// TwinCAT 3 PLC project XtsTransport
// Title: XTS Transport
// Author: HAUD
// ProjectVersion: 4.01.02
// Description: . XTS_TRANSPORT_LAYER by Daniel Hauer
// ProgramVersion: 3.1.4026.26
// libraries:
//   Tc2_EtherCAT, * (Beckhoff Automation GmbH)
//   Tc2_Math, * (Beckhoff Automation GmbH)
//   Tc2_MC2, * (Beckhoff Automation GmbH)
//   Tc2_Standard, * (Beckhoff Automation GmbH)
//   Tc2_System, * (Beckhoff Automation GmbH)
//   Tc2_Utilities, * (Beckhoff Automation GmbH)
//   Tc2_XmlDataSrv, * (Beckhoff Automation GmbH)
//   Tc3_McCollisionAvoidance, * (Beckhoff Automation GmbH)
//   Tc3_McCoordinatedMotion, * (Beckhoff Automation GmbH)
//   Tc3_Module, * (Beckhoff Automation GmbH)
//   Tc3_XTS_Utility, * (Beckhoff Automation GmbH)
//   VisuDialogs, * (System)
// project tree:
//   APPLICATION/ GVL_APPLICATION.TcGVL (not stored), MAIN_APP.TcPOU, StationParameterExample.TcPOU, XTS_TRANSPORT_1.TcVIS (not stored)
//   APPLICATION/_config/ StationParameterExample.TcPOU (not stored)
//   APPLICATION/_types/Application/ E_APP_CHECK.TcDUT (not stored), E_APP_VARIANT.TcDUT (not stored), ST_APP_CTRL.TcDUT (not stored), ST_APP_STATE.TcDUT (not stored)
//   APPLICATION/_types/Collector/ E_PROCESS_CHECK.TcDUT (not stored), E_PROCESS_CTRL.TcDUT (not stored), E_PROCESS_STATE.TcDUT (not stored), fb_ProcessCollector.TcPOU (not stored), fb_StationCollector.TcPOU (not stored), I_ProcessCollector.TcIO (not stored), ST_PROCESS_CTRL.TcDUT (not stored), ST_PROCESS_STATE.TcDUT (not stored), T_PROCESS.TcDUT
//   APPLICATION/_types/ fb_ProcessConductor.TcPOU (not stored)
//   APPLICATION/_types/Instance/ E_INSTANCE.TcDUT (not stored), E_INSTANCE_CHECK.TcDUT (not stored), E_INSTANCE_CMD.TcDUT (not stored), E_INSTANCE_STATE.TcDUT (not stored), fb_Instance.TcPOU (not stored), ST_INSTANCE_CTRL.TcDUT (not stored), ST_INSTANCE_STATE.TcDUT (not stored)
//   APPLICATION/_types/LinkedList/ E_LIST_CHECK.TcDUT (not stored), E_LIST_CTRL.TcDUT (not stored), E_LIST_STATE.TcDUT (not stored), fb_Process_LinkedList.TcPOU (not stored), fb_Process_LinkedListCtrl.TcPOU (not stored), I_Process_LinkedList.TcIO (not stored), ST_LIST_CTRL.TcDUT (not stored), ST_LIST_NODE_DATA.TcDUT (not stored), ST_LIST_STATE.TcDUT (not stored), ST_PROCESS_DATA.TcDUT (not stored), ST_PROCESS_LIST_RESULT.TcDUT (not stored)
//   / GlobalTextList.TcGTLO, PlcTask.TcTTO
//   MAPPING/ MAPPING_XTS_in.TcPOU, MAPPING_XTS_out.TcPOU (not stored)
//   MAPPING/_types/ E_MAPPING_CHECK.TcDUT (not stored), U_APP_CTRL.TcDUT (not stored), U_APP_STATE.TcDUT (not stored), U_GEAR_DATA.TcDUT (not stored), U_INSTANCE_CTRL.TcDUT (not stored), U_INSTANCE_STATE.TcDUT (not stored), U_MOVER_CTRL.TcDUT (not stored), U_MOVER_INFO.TcDUT (not stored), U_MOVER_SELECTOR_CTRL.TcDUT (not stored), U_MOVER_SELECTOR_STATE.TcDUT (not stored), U_MOVER_STATE.TcDUT (not stored), U_MOVE_DATA.TcDUT (not stored), U_TICKET_LIST_CTRL.TcDUT (not stored), U_TICKET_LIST_DATA_INPUT.TcDUT (not stored), U_TICKET_LIST_DATA_OUTPUT.TcDUT (not stored), U_TICKET_LIST_STATE.TcDUT (not stored), U_XTS_STATION_CTRL.TcDUT (not stored), U_XTS_STATION_STATE.TcDUT (not stored), U_XTS_TRANSPORT_CTRL.TcDUT (not stored), U_XTS_TRANSPORT_STATE.TcDUT (not stored)
//   PLC_MOTION/_GVL/ PLC_CONSTANT.TcGVL
//   XTS_TRANSPORT/CaGroup/ FB_CaGroup.TcPOU (not stored), I_XtsTransport_CaGroup.TcIO (not stored)
//   XTS_TRANSPORT/CaGroup/types/ E_CA_GROUP_STATE.TcDUT, E_GROUP_CHECK.TcDUT, ST_GROUP_INFO.TcDUT
//   XTS_TRANSPORT/ GVL_XTS.TcGVL (not stored), GVL_XTS_CONSTANTS.TcGVL, GVL_XTS_VERSION.TcGVL (not stored), MAIN_XTS.TcPOU (not stored)
//   XTS_TRANSPORT/Mover/ fb_Mover.TcPOU (not stored), fb_MoverCtrl.TcPOU (not stored), fb_MoverSelector.TcPOU (not stored), I_XtsTransport_Mover.TcIO (not stored)
//   XTS_TRANSPORT/Mover/types/ E_MOVER_CHECK.TcDUT, E_MOVER_CTRL.TcDUT, E_MOVER_SELECTOR.TcDUT, E_MOVER_STATE.TcDUT, ST_GEAR_DATA.TcDUT, ST_MOVER_CTRL.TcDUT, ST_MOVER_INFO.TcDUT, ST_MOVER_SELECTOR_CTRL.TcDUT, ST_MOVER_SELECTOR_STATE.TcDUT, ST_MOVER_STATE.TcDUT, ST_MOVE_DATA.TcDUT
//   XTS_TRANSPORT/Xpu/ fb_Xpu.TcPOU (not stored), fb_XpuCtrl.TcPOU (not stored), I_XtsTransport_Xpu.TcIO (not stored)
//   XTS_TRANSPORT/Xpu/types/ E_XPU_CHECK.TcDUT, E_XPU_CTRL.TcDUT, E_XPU_INIT.TcDUT, E_XPU_STATE.TcDUT, ST_XPU_CTRL.TcDUT, ST_XPU_INFO.TcDUT, ST_XPU_STATE.TcDUT
//   XTS_TRANSPORT/XtsStation/ fb_StationGearInPos.TcPOU (not stored), fb_StationProcess.TcPOU (not stored), I_XtsTransport_Station.TcIO (not stored)
//   XTS_TRANSPORT/XtsStation/types/ E_STATION_CHECK.TcDUT, E_STATION_CTRL.TcDUT, E_STATION_GEAR_DISTANCE_AXIS.TcDUT, E_STATION_STATE.TcDUT, E_STATION_TYPE.TcDUT, fb_StationBase.TcPOU (not stored), fb_Station_LinkedList.TcPOU (not stored), I_Station_LinkedList.TcIO (not stored), ST_STATION_CTRL.TcDUT, ST_STATION_GEAR_PARAMETER.TcDUT, ST_STATION_LIST_RESULT.TcDUT, ST_STATION_MOVER_DATA.TcDUT, ST_STATION_PARAMETER.TcDUT, ST_STATION_STATE.TcDUT, T_NEST_OFFSET.TcDUT
//   XTS_TRANSPORT/XtsTransportUnit/ fb_TransportUnit.TcPOU (not stored)
//   XTS_TRANSPORT/XtsTransportUnit/types/ E_XTS_TRANSPORT_CHECK.TcDUT, E_XTS_TRANSPORT_CTRL.TcDUT, E_XTS_TRANSPORT_STATE.TcDUT, ST_XTS_TRANSPORT_CTRL.TcDUT, ST_XTS_TRANSPORT_STATE.TcDUT
//   XTS_TRANSPORT/_Visualization/ GROUP_VISU.TcVIS, MOVER_VISU.TcVIS, SELECTOR_VISU.TcVIS, STATION_VISU.TcVIS, Visualization Manager.TcVMO (not stored), XPU_VISU.TcVIS, XTS_TRANSPORT.TcVIS (not stored)
//   XTS_TRANSPORT/_Visualization/textlists/ TL_E_CTRL_MOVER.TcTLO, TL_E_CTRL_STATION.TcTLO, TL_E_CTRL_TRANSPORT.TcTLO, TL_E_CTRL_XPU.TcTLO, TL_E_MOVER_SELECTOR.TcTLO (not stored)
//   XTS_TRANSPORT/_Visualization/types/ ST_XPU_STRINGS.TcDUT, T_MOVER_SELECTOR.TcVIS
//   _MSG/class/ fb_LocalTime.TcPOU (not stored), fb_MessageData.TcPOU (not stored), fb_MessageDataCtrl.TcPOU
//   _MSG/ f_MessageSet.TcPOU (not stored), GVL_MSG_AXIS.TcGVL (not stored), GVL_MSG_XTS.TcGVL, I_MessageData.TcIO
//   _MSG/types/ e_Device.TcDUT, E_MessageType.TcDUT, E_MESSAGE_BATCH.TcDUT, E_MESSAGE_CHECK.TcDUT, E_MESSAGE_CTRL.TcDUT, E_MESSAGE_FLOW.TcDUT, E_MESSAGE_STATE.TcDUT, e_Subdevice.TcDUT, ST_Message.TcDUT, ST_MESSAGE_CTRL.TcDUT, ST_MESSAGE_STATE.TcDUT, TL_E_MESSAGETYPE.TcTLO
//   _types/ E_CHECK_STATE.TcDUT (not stored), E_PROGRESS.TcDUT (not stored), f_GetProgress.TcPOU (not stored), f_GetState.TcPOU (not stored), T_PROCESS.TcDUT (not stored)
//   _XML/Configuration/ fb_Configuration.TcPOU (not stored), I_Configuration_Station.TcIO (not stored)
//   _XML/Configuration/types/ ST_Configuration.TcDUT
//   _XML/ fb_XmlBase.TcPOU (not stored)
//   _XML/PositionOffsets/ fb_MoverPositionOffsetData.TcPOU (not stored)
//   _XML/PositionOffsets/types/ ST_MOVER_OFFSETS.TcDUT
//   _XML/types/ E_DATA_CHECK.TcDUT, E_DATA_CTRL.TcDUT, E_DATA_STATE.TcDUT, fb_XmlRead.TcPOU, fb_XmlWrite.TcPOU, ST_DATA_CTRL.TcDUT, ST_DATA_STATE.TcDUT
// (motion and I/O tree: see PLC project externcontrol)
// real-time tasks:
//   TASK XTS Task 1: cycle T#250us, priority 1, ADS port 350
//   TASK XTS Task 2: cycle T#250us, priority 3, ADS port 352
//   TASK PlcTask: cycle T#1ms, priority 15, ADS port 353
//   TASK Job Task: cycle default, priority 32
// variable links:
//   ExternControl/ExternControl Instance <-> XtsTransport/XtsTransport Instance
//     PlcTask Inputs/MAIN_APP.eInitXtsTransport <-> PlcTask Outputs/MAIN_APP.eInit
//     PlcTask Inputs/MAPPING_in.StationState.byState <-> PlcTask Outputs/MAPPING_XTS_out.StationState.byState
//     PlcTask Inputs/MAPPING_in.TransportState.byState <-> PlcTask Outputs/MAPPING_XTS_out.TransportState.byState
//     PlcTask Outputs/MAPPING_out.StationControl.byCtrl <-> PlcTask Inputs/MAPPING_XTS_in.StationControl.byCtrl
//     PlcTask Outputs/MAPPING_out.TransportControl.byCtrl <-> PlcTask Inputs/MAPPING_XTS_in.TransportControl.byCtrl
//   XtsTransport/XtsTransport Instance <-> NC-Task 1/Axes/Mover Axis 1
//     PlcTask Inputs/GVL_XTS.AxisRefMover[1].NcToPlc <-> Outputs/ToPlc
//     PlcTask Outputs/GVL_XTS.AxisRefMover[1].PlcToNc <-> Inputs/FromPlc
//   XtsTransport/XtsTransport Instance <-> NC-Task 1/Axes/Mover Axis 10
//     PlcTask Inputs/GVL_XTS.AxisRefMover[10].NcToPlc <-> Outputs/ToPlc
//     PlcTask Outputs/GVL_XTS.AxisRefMover[10].PlcToNc <-> Inputs/FromPlc
//   XtsTransport/XtsTransport Instance <-> NC-Task 1/Axes/Mover Axis 11
//     PlcTask Inputs/GVL_XTS.AxisRefMover[11].NcToPlc <-> Outputs/ToPlc
//     PlcTask Outputs/GVL_XTS.AxisRefMover[11].PlcToNc <-> Inputs/FromPlc
//   XtsTransport/XtsTransport Instance <-> NC-Task 1/Axes/Mover Axis 12
//     PlcTask Inputs/GVL_XTS.AxisRefMover[12].NcToPlc <-> Outputs/ToPlc
//     PlcTask Outputs/GVL_XTS.AxisRefMover[12].PlcToNc <-> Inputs/FromPlc
//   XtsTransport/XtsTransport Instance <-> NC-Task 1/Axes/Mover Axis 13
//     PlcTask Inputs/GVL_XTS.AxisRefMover[13].NcToPlc <-> Outputs/ToPlc
//     PlcTask Outputs/GVL_XTS.AxisRefMover[13].PlcToNc <-> Inputs/FromPlc
//   XtsTransport/XtsTransport Instance <-> NC-Task 1/Axes/Mover Axis 14
//     PlcTask Inputs/GVL_XTS.AxisRefMover[14].NcToPlc <-> Outputs/ToPlc
//     PlcTask Outputs/GVL_XTS.AxisRefMover[14].PlcToNc <-> Inputs/FromPlc
//   XtsTransport/XtsTransport Instance <-> NC-Task 1/Axes/Mover Axis 15
//     PlcTask Inputs/GVL_XTS.AxisRefMover[15].NcToPlc <-> Outputs/ToPlc
//     PlcTask Outputs/GVL_XTS.AxisRefMover[15].PlcToNc <-> Inputs/FromPlc
//   XtsTransport/XtsTransport Instance <-> NC-Task 1/Axes/Mover Axis 16
//     PlcTask Inputs/GVL_XTS.AxisRefMover[16].NcToPlc <-> Outputs/ToPlc
//     PlcTask Outputs/GVL_XTS.AxisRefMover[16].PlcToNc <-> Inputs/FromPlc
//   XtsTransport/XtsTransport Instance <-> NC-Task 1/Axes/Mover Axis 17
//     PlcTask Inputs/GVL_XTS.AxisRefMover[17].NcToPlc <-> Outputs/ToPlc
//     PlcTask Outputs/GVL_XTS.AxisRefMover[17].PlcToNc <-> Inputs/FromPlc
//   XtsTransport/XtsTransport Instance <-> NC-Task 1/Axes/Mover Axis 18
//     PlcTask Inputs/GVL_XTS.AxisRefMover[18].NcToPlc <-> Outputs/ToPlc
//     PlcTask Outputs/GVL_XTS.AxisRefMover[18].PlcToNc <-> Inputs/FromPlc
//   XtsTransport/XtsTransport Instance <-> NC-Task 1/Axes/Mover Axis 19
//     PlcTask Inputs/GVL_XTS.AxisRefMover[19].NcToPlc <-> Outputs/ToPlc
//     PlcTask Outputs/GVL_XTS.AxisRefMover[19].PlcToNc <-> Inputs/FromPlc
//   XtsTransport/XtsTransport Instance <-> NC-Task 1/Axes/Mover Axis 2
//     PlcTask Inputs/GVL_XTS.AxisRefMover[2].NcToPlc <-> Outputs/ToPlc
//     PlcTask Outputs/GVL_XTS.AxisRefMover[2].PlcToNc <-> Inputs/FromPlc
//   XtsTransport/XtsTransport Instance <-> NC-Task 1/Axes/Mover Axis 20
//     PlcTask Inputs/GVL_XTS.AxisRefMover[20].NcToPlc <-> Outputs/ToPlc
//     PlcTask Outputs/GVL_XTS.AxisRefMover[20].PlcToNc <-> Inputs/FromPlc
//   XtsTransport/XtsTransport Instance <-> NC-Task 1/Axes/Mover Axis 21
//     PlcTask Inputs/GVL_XTS.AxisRefMover[21].NcToPlc <-> Outputs/ToPlc
//     PlcTask Outputs/GVL_XTS.AxisRefMover[21].PlcToNc <-> Inputs/FromPlc
//   XtsTransport/XtsTransport Instance <-> NC-Task 1/Axes/Mover Axis 22
//     PlcTask Inputs/GVL_XTS.AxisRefMover[22].NcToPlc <-> Outputs/ToPlc
//     PlcTask Outputs/GVL_XTS.AxisRefMover[22].PlcToNc <-> Inputs/FromPlc
//   XtsTransport/XtsTransport Instance <-> NC-Task 1/Axes/Mover Axis 23
//     PlcTask Inputs/GVL_XTS.AxisRefMover[23].NcToPlc <-> Outputs/ToPlc
//     PlcTask Outputs/GVL_XTS.AxisRefMover[23].PlcToNc <-> Inputs/FromPlc
//   XtsTransport/XtsTransport Instance <-> NC-Task 1/Axes/Mover Axis 24
//     PlcTask Inputs/GVL_XTS.AxisRefMover[24].NcToPlc <-> Outputs/ToPlc
//     PlcTask Outputs/GVL_XTS.AxisRefMover[24].PlcToNc <-> Inputs/FromPlc
//   XtsTransport/XtsTransport Instance <-> NC-Task 1/Axes/Mover Axis 25
//     PlcTask Inputs/GVL_XTS.AxisRefMover[25].NcToPlc <-> Outputs/ToPlc
//     PlcTask Outputs/GVL_XTS.AxisRefMover[25].PlcToNc <-> Inputs/FromPlc
//   XtsTransport/XtsTransport Instance <-> NC-Task 1/Axes/Mover Axis 26
//     PlcTask Inputs/GVL_XTS.AxisRefMover[26].NcToPlc <-> Outputs/ToPlc
//     PlcTask Outputs/GVL_XTS.AxisRefMover[26].PlcToNc <-> Inputs/FromPlc
//   XtsTransport/XtsTransport Instance <-> NC-Task 1/Axes/Mover Axis 27
//     PlcTask Inputs/GVL_XTS.AxisRefMover[27].NcToPlc <-> Outputs/ToPlc
//     PlcTask Outputs/GVL_XTS.AxisRefMover[27].PlcToNc <-> Inputs/FromPlc
//   XtsTransport/XtsTransport Instance <-> NC-Task 1/Axes/Mover Axis 28
//     PlcTask Inputs/GVL_XTS.AxisRefMover[28].NcToPlc <-> Outputs/ToPlc
//     PlcTask Outputs/GVL_XTS.AxisRefMover[28].PlcToNc <-> Inputs/FromPlc
//   XtsTransport/XtsTransport Instance <-> NC-Task 1/Axes/Mover Axis 3
//     PlcTask Inputs/GVL_XTS.AxisRefMover[3].NcToPlc <-> Outputs/ToPlc
//     PlcTask Outputs/GVL_XTS.AxisRefMover[3].PlcToNc <-> Inputs/FromPlc
//   XtsTransport/XtsTransport Instance <-> NC-Task 1/Axes/Mover Axis 4
//     PlcTask Inputs/GVL_XTS.AxisRefMover[4].NcToPlc <-> Outputs/ToPlc
//     PlcTask Outputs/GVL_XTS.AxisRefMover[4].PlcToNc <-> Inputs/FromPlc
//   XtsTransport/XtsTransport Instance <-> NC-Task 1/Axes/Mover Axis 5
//     PlcTask Inputs/GVL_XTS.AxisRefMover[5].NcToPlc <-> Outputs/ToPlc
//     PlcTask Outputs/GVL_XTS.AxisRefMover[5].PlcToNc <-> Inputs/FromPlc
//   XtsTransport/XtsTransport Instance <-> NC-Task 1/Axes/Mover Axis 6
//     PlcTask Inputs/GVL_XTS.AxisRefMover[6].NcToPlc <-> Outputs/ToPlc
//     PlcTask Outputs/GVL_XTS.AxisRefMover[6].PlcToNc <-> Inputs/FromPlc
//   XtsTransport/XtsTransport Instance <-> NC-Task 1/Axes/Mover Axis 7
//     PlcTask Inputs/GVL_XTS.AxisRefMover[7].NcToPlc <-> Outputs/ToPlc
//     PlcTask Outputs/GVL_XTS.AxisRefMover[7].PlcToNc <-> Inputs/FromPlc
//   XtsTransport/XtsTransport Instance <-> NC-Task 1/Axes/Mover Axis 8
//     PlcTask Inputs/GVL_XTS.AxisRefMover[8].NcToPlc <-> Outputs/ToPlc
//     PlcTask Outputs/GVL_XTS.AxisRefMover[8].PlcToNc <-> Inputs/FromPlc
//   XtsTransport/XtsTransport Instance <-> NC-Task 1/Axes/Mover Axis 9
//     PlcTask Inputs/GVL_XTS.AxisRefMover[9].NcToPlc <-> Outputs/ToPlc
//     PlcTask Outputs/GVL_XTS.AxisRefMover[9].PlcToNc <-> Inputs/FromPlc
//   XtsTransport/XtsTransport Instance <-> NC-Task 1/Objects/Group1 (CA Group)
//     PlcTask Inputs/GVL_XTS.CaGroupRef.NcToPlc/CA <-> Group Outputs/ToPLC
//     PlcTask Outputs/GVL_XTS.CaGroupRef.PlcToNc/CA <-> Group Inputs/FromPLC

CONFIGURATION XtsTransport
    RESOURCE PLC ON TwinCAT3
        TASK PlcTask(INTERVAL := T#1ms, PRIORITY := 15);
        PROGRAM MAPPING_in WITH PlcTask : MAPPING_in;
        PROGRAM MAIN WITH PlcTask : MAIN;
        PROGRAM MAPPING_out WITH PlcTask : MAPPING_out;
    END_RESOURCE
END_CONFIGURATION

// ---- APPLICATION/_types/Collector/T_PROCESS.TcDUT
TYPE T_PROCESS : DWORD; END_TYPE

// ---- XTS_TRANSPORT/CaGroup/types/E_CA_GROUP_STATE.TcDUT
// {attribute 'qualified_only'}
// {attribute 'strict'}
{attribute 'to_string'}
TYPE E_CA_GROUP_STATE :
(
  // replicated from MC_GROUP_STATE for getting to_string() functionality
	mcGroupStateInvalid   :=0, 
  mcGroupStateDisabled  :=1, 
  mcGroupStateStandby   :=2, 
  mcGroupStateMoving    :=3, 
  mcGroupStateStopping  :=4, 
  mcGroupStateErrorStop :=5, 
  mcGroupStateHoming    :=6, 
  mcGroupStateNotReady  :=7, 
  mcGroupStateSuspended :=8 
)UINT;
END_TYPE

// ---- XTS_TRANSPORT/CaGroup/types/E_GROUP_CHECK.TcDUT
{attribute 'qualified_only'}
{attribute 'to_string'}
TYPE E_GROUP_CHECK :
(
  NULL,
  REFERENCE_GROUP_REF_INVALID := 9000,
  REFERENCE_AXIS_REF_INVALID,
  REFERENCE_CTRL_INVALID,
  REFERENCE_STATE_INVALID,
  REFERENCE_MOVER_ITF_INVALID,
  REFERENCE_XPU_INFO_INVALID,

  CHECK_DONE              := 10000
)UINT;
END_TYPE

// ---- XTS_TRANSPORT/CaGroup/types/ST_GROUP_INFO.TcDUT
TYPE ST_GROUP_INFO :
STRUCT
  GroupStatusValid,
  GroupStatusBusy,
  GroupMoving, 
  GroupHoming, 
  GroupErrorStop, 
  GroupNotReady, 
  GroupStandby, 
  GroupStopping,
 
  GroupDisabled, 
  AllAxesStanding, 
  ConstantVelocity, 
  Accelerating, 
  Decelerating, 
  InPosition, 
  GroupError					  : BIT; 

  GroupErrorId					: UDINT;

  AxisCount      				: UDINT;
  AxisCountEnabled      : UDINT;

  {attribute 'displaymode':='hex'}
  CaGroupOID            : OTCID;

  CaGroupState          : E_CA_GROUP_STATE;
END_STRUCT
END_TYPE

// ---- XTS_TRANSPORT/Mover/types/E_MOVER_CHECK.TcDUT
{attribute 'qualified_only'}
{attribute 'strict'}
{attribute 'to_string'}
TYPE E_MOVER_CHECK :
(
  NULL,
  MOVER_ID_INVALID := 9000,
  REFERENCE_AXIS_REF_INVALID,
  REFERENCE_LAST_POSITION_INVALID,
  REFERENCE_LAST_GAP_INVALID,
  REFERENCE_INFO_INVALID,

  REFERENCE_CTRL_INVALID  := 9100,
  REFERENCE_STATE_INVALID,
  REFERENCE_GEAR_DATA_INVALID,
  REFERENCE_MOVE_DATA_INVALID,
  REFERENCE_MOVER_ITF_INVALID,

  CHECK_DONE  := 10_000
)UINT;
END_TYPE

// ---- XTS_TRANSPORT/Mover/types/E_MOVER_CTRL.TcDUT
{attribute 'qualified_only'}
{attribute 'strict'}
{attribute 'to_string'}
TYPE E_MOVER_CTRL :
(
  MOVER_NULL,               // initial value at startup, used for change of order or retrigger
  MOVER_ENABLE,             // sets MC_Power.Enable
  MOVER_DISABLE,            // removes MC_Power.Enable
  MOVER_MOVE_TO_POS,        // modulo absolute positioning with MC_MoveAbsolute, InTargetPosition check
  MOVER_MOVE_TO_POS_CA,     // modulo absolute positioning with MC_MoveAbsoluteCA, InTargetPosition check
  MOVER_SEND_TO_POS_CA,     // modulo absolute positioning with MC_MoveAbsoluteCA, done after moving ReleaseDistance
  MOVER_HALT,               // halts mover; by use of MC_Halt mover is set passive in CA group
  MOVER_GEAR_IN,            // GearIn for mover in standstill

  MOVER_GEAR_IN_POS_CA,     // GearInPosCA of mover; when FB_GearInPosCa is InSync --> order is done; check SyncDistance yourself and release mover with e_mover_order.mover_SendToPos
  MOVER_GEAR_OUT,           // gear out for mover
  MOVER_RESET,              // MC_RESET for mover
  MOVER_INFO                // used to display MoverInfo in ST_MOVER_SELECTOR_STATE.Info
)UINT;
END_TYPE

// ---- XTS_TRANSPORT/Mover/types/E_MOVER_SELECTOR.TcDUT
{attribute 'qualified_only'}
{attribute 'strict'}
{attribute 'to_string'}
TYPE E_MOVER_SELECTOR :
(
	SELECT_MOVER_INDEX,
  SELECT_MOVER_AXIS_ID
);
END_TYPE

// ---- XTS_TRANSPORT/Mover/types/E_MOVER_STATE.TcDUT
{attribute 'qualified_only'}
{attribute 'to_string'}
TYPE E_MOVER_STATE :
(
  MOVER_NULL,               // initial value at startup, used for change of order or retrigger
  MOVER_ENABLE,             // sets MC_Power.Enable
  MOVER_DISABLE,            // removes MC_Power.Enable
  MOVER_MOVE_TO_POS,        // modulo absolute positioning with MC_MoveAbsolute, InTargetPosition check
  MOVER_MOVE_TO_POS_CA,     // modulo absolute positioning with MC_MoveAbsoluteCA, InTargetPosition check
  MOVER_SEND_TO_POS_CA,     // modulo absolute positioning with MC_MoveAbsoluteCA, done after moving ReleaseDistance
  MOVER_HALT,               // halts mover; by use of MC_Halt mover is set passive in CA group
  MOVER_GEAR_IN,            // GearIn for mover in standstill

  MOVER_GEAR_IN_POS_CA,     // GearInPosCA of mover; when FB_GearInPosCa is InSync --> order is done; check SyncDistance yourself and release mover with e_mover_order.mover_SendToPos
  MOVER_GEAR_OUT,           // gear out for mover
  MOVER_RESET,              // MC_RESET for mover
  MOVER_INFO
)UINT;
END_TYPE

// ---- XTS_TRANSPORT/Mover/types/ST_GEAR_DATA.TcDUT
{attribute 'pack_mode' := '2'}
TYPE ST_GEAR_DATA :
STRUCT
  rDeltaToMasterPos       : LREAL;
  rModuloSyncPosSlave     : LREAL;
  rMasterStartDistance    : LREAL;
  rGearNumerator          : LREAL;
  iGearDenumerator        : USINT  := 1;
END_STRUCT
END_TYPE

// ---- XTS_TRANSPORT/Mover/types/ST_MOVER_CTRL.TcDUT
{attribute 'pack_mode' := '2'}
TYPE ST_MOVER_CTRL :
STRUCT
  Cmd             : E_MOVER_CTRL;  // order to execute on mover
END_STRUCT
END_TYPE

// ---- XTS_TRANSPORT/Mover/types/ST_MOVER_INFO.TcDUT
{attribute 'pack_mode' := '2'}
TYPE ST_MOVER_INFO :
STRUCT
  bMoverEnabled           : BIT;    // Axis[i].Status.ControlLoopClosed
  bMoverError             : BIT;    // Axis[i].Status.Error
  bMoverCoupled           : BIT;    // Axis[i].Status.Coupled OR _fbGearInPosCa[i].InSync
  bMoverStandstill        : BIT;    // Axis[i].Status.NotMoving
  bMoverAvoidingCollision : BIT;    // Axis[i].NcToPlc.StateDWord2.0
  bMoverInTarget          : BIT;    // Axis[i].NcToPlc.ActPos == rLastSetPos[i]

  rModuloActPos           : LREAL;  // Axis[i].NcToPlc.ModuloActPos
  rAbsActPos              : LREAL;  // Axis[i].NcToPlc.ActPos
  rAbsTargetPos           : LREAL;  // rLastSetPos[i]
  rModuloTargetPos        : LREAL;  // Tc2_Math.LMOD(_rLastSetPos[i], _RailLength)

  nErrorId                : UDINT;
END_STRUCT
END_TYPE

// ---- XTS_TRANSPORT/Mover/types/ST_MOVER_SELECTOR_CTRL.TcDUT
TYPE ST_MOVER_SELECTOR_CTRL :
STRUCT
  Selector      : E_MOVER_SELECTOR; // select by array Index OR AXIS_REF.NcToPlc.AxisId 
  Mover         : UINT;             // array Index OR AXIS_REF.NcToPlc.AxisId
  Control       : ST_MOVER_CTRL;    // mover control struct, put motion command in here

  Data          : ST_MOVE_DATA;     // write your movement parameters
  //Gear          : ST_GEAR_DATA;     // write your gearing parameters
END_STRUCT
END_TYPE

// ---- XTS_TRANSPORT/Mover/types/ST_MOVER_SELECTOR_STATE.TcDUT
TYPE ST_MOVER_SELECTOR_STATE :
STRUCT
  MoverIndex  : UINT;
  AxisId      : UDINT;
  State       : ST_MOVER_STATE;

  Info        : ST_MOVER_INFO;
END_STRUCT
END_TYPE

// ---- XTS_TRANSPORT/Mover/types/ST_MOVER_STATE.TcDUT
{attribute 'pack_mode' := '2'}
TYPE ST_MOVER_STATE :
STRUCT
  State           : E_MOVER_STATE;  // ST_MOVER_CTRL.Cmd with added E_PROGRESS
  MasterId        : USINT;            // mirror NC AxisId of Master axis
END_STRUCT
END_TYPE

// ---- XTS_TRANSPORT/Mover/types/ST_MOVE_DATA.TcDUT
{attribute 'pack_mode' := '2'}
TYPE ST_MOVE_DATA :
STRUCT
  // HAUD 2024 03 14
  // some init data added for example
  rPos            : LREAL :=   2275.0;
  rVelo           : LREAL :=    500.0;
  rAcc            : LREAL :=   5000.0;
  rJerk           : LREAL := 500000.0;
  rGap            : LREAL :=    100.0;
  rOverride       : LREAL :=    100.0;
  rDelta          : LREAL :=      0.05;
  rDistance       : LREAL :=     25.0;
END_STRUCT
END_TYPE

// ---- XTS_TRANSPORT/Xpu/types/E_XPU_CHECK.TcDUT
{attribute 'qualified_only'}
{attribute 'to_string'}
TYPE E_XPU_CHECK :
(
  INIT_CHECK,
  INIT_CHECK_ERROR,
  START_CHECK,
  XPU_INSTANCE_NULL,
  XPU_RAIL_LENGTH,
  GROUP_RAIL_LENGTH,
  RAIL_LENGTH_COMPARE,
  GROUP_NOT_CONFIGURED,
  GROUP_OID_MISMATCH,

  MOVER_COUNT             := 10,
  MOVER_COUNT_ZERO,
  MOVER_COUNT_NOT_EQUAL,

  PROCESSING_UNIT_POSITIONS_VALID         := 20,
  PROCESSING_UNIT_GET_DATA_EXCEED,

  MOVER_ID_STANDARD       := 30,
  MOVER_ID_SIMULATION,
  MOVER_ID_DETECTION_MODE,
  MOVER_ID_DETECTION_VALID,
  MOVER_ID_DETECTION_DC_LINK,
  MOVER_ID_DETECTION_BUSY,
  MOVER_ID_DETECTION_IDLE,
  MOVER_ID_DETECTION_STATE,
  MOVER_ID_MULTIPLE_NOT_SUPPORTED,

  POINTER_CHECK           := 90,
  POINTER_NULL_CTRL,
  POINTER_NULL_STATE,

  CHECK_DONE      := 10_000
)UINT;
END_TYPE

// ---- XTS_TRANSPORT/Xpu/types/E_XPU_CTRL.TcDUT
{attribute 'strict'}
TYPE E_XPU_CTRL :
(
  XTS_CMD_NULL,
  XTS_CMD_INIT                  := 10,
  //XTS_CMD_READ_STN_CONFIG       := 20,
  XTS_IDLE                      := 30
)UINT;
END_TYPE

// ---- XTS_TRANSPORT/Xpu/types/E_XPU_INIT.TcDUT
{attribute 'to_string'}
TYPE E_XPU_INIT :
(
	INIT_START,
  INIT_ENVIRONMENT_OID            := 10,
  INIT_INFO_SERVER_ITF,
  INIT_INFO_SERVER_STATION_COUNT,
  INIT_INFO_SERVER_STATION_OID,
  INIT_CA_GROUP_OID               := 20,
  INIT_CA_GROUP_GET_OID,
  INIT_CA_GROUP_CHECK_OID,
  INIT_CA_GROUP_COM,
  INIT_PARAMETERSET_COUNT,
  INIT_PARAMETERSET_OID,
  INIT_PARAMETERSET_COM,
  INIT_PARAMETERSET_COM_INIT,
  INIT_PARAMETERSET_COM_NEXT,
  INIT_PROCESSING_UNIT_COM        := 30,
  INIT_PROCESSING_UNIT_COM_INIT,
  INIT_PROCESSING_UNIT_PART_COUNT,
  INIT_PROCESSING_UNIT_PART_OID,
  INIT_PROCESSING_UNIT_TRACK_COUNT,
  INIT_PROCESSING_UNIT_TRACK_OID,
  INIT_PROCESSING_UNIT_MOVER_COUNT,
  INIT_PROCESSING_UNIT_MOVER_OID,
  INIT_PROCESSING_UNIT_TASK_COUNT,
  INIT_PROCESSING_UNIT_TASK_OID,
  INIT_TRACK_COM                  := 50,
  INIT_TRACK_COM_INIT,
  INIT_PART_COM                   := 60,
  INIT_PART_COM_INIT,
  INIT_PART_MODULE_COUNT,
  INIT_PART_MODULE_OID,
  INIT_PART_MODULE_COM,
  INIT_PART_MODULE_COM_INIT,
  INIT_PART_MODULE_COM_NEXT,
  INIT_MOVER_COM                  := 70,
  INIT_MOVER_COM_INIT,
  INIT_MOVER_COM_NEXT,
  INIT_NCT_CONTROLLER_OID         := 80,
  INIT_NCT_CONTROLLER_COM,
  INIT_NCT_CONTROLLER_COM_INIT,
  INIT_NCT_BASE_UNIT_COUNT,
  INIT_NCT_BASE_UNIT_ITF,
  INIT_NCT_BASE_UNIT_NEXT,
  INIT_DATA_GET                   := 90,
  INIT_DATA_CHECK,
  INIT_DONE                       := 100
)UINT;
END_TYPE

// ---- XTS_TRANSPORT/Xpu/types/E_XPU_STATE.TcDUT
{attribute 'to_string'}
TYPE E_XPU_STATE :
(
  XTS_NULL,
  XTS_INVALID,
  XTS_INIT                      := 10,    // initialize XPU
  XTS_STATION_INFO_READ         := 20,    // get Station information from Xpu
  XTS_IDLE                      := 30
)UINT;
END_TYPE

// ---- XTS_TRANSPORT/Xpu/types/ST_XPU_CTRL.TcDUT
{attribute 'pack_mode' := '2'}
TYPE ST_XPU_CTRL :
STRUCT
  Cmd             : E_XPU_CTRL;
END_STRUCT
END_TYPE

// ---- XTS_TRANSPORT/Xpu/types/ST_XPU_INFO.TcDUT
{attribute 'pack_mode' := '2'}
TYPE ST_XPU_INFO :
STRUCT
  AllPositionsValid   : BIT;
  IdDetectionError    : BIT;
  IdDetectionValid    : BIT;
  IdDetectionActive   : BIT;

  OperationMode       : UINT;

  IdDetectionMode           : UINT;
  MoverPositionAssignement  : UINT;

  nDetectedAxisCount  : UINT;
  nExpectedAxisCount  : UINT;

  nParameterSetCount  : UINT;
  nModuleCount        : UINT;
  rRailLength         : LREAL;
END_STRUCT
END_TYPE

// ---- XTS_TRANSPORT/Xpu/types/ST_XPU_STATE.TcDUT
{attribute 'pack_mode' := '2'}
TYPE ST_XPU_STATE :
STRUCT
  Init            : E_XPU_INIT;
  State           : E_XPU_STATE;
  Check           : E_XPU_CHECK;  // cyclic check result
  DcLink          : BIT;          // power all motor modules is ON
END_STRUCT
END_TYPE

// ---- XTS_TRANSPORT/XtsStation/types/E_STATION_CHECK.TcDUT
{attribute 'qualified_only'}
{attribute 'strict'}
{attribute 'to_string'}
TYPE E_STATION_CHECK :
(
	CHECK_NULL,
  STATION_ID_INVALID := 9000,
  REFERENCE_CTRL_INVALID,
  REFERENCE_STATE_INVALID,
  REFERENCE_LIST_ITF_INVALID,
  REFERENCE_MOVER_ITF_INVALID,
  REFERENCE_MOVER_OFFSET_INVALID,
  REFERENCE_PARAMETER_INVALID,
  REFERENCE_MOVER_AXIS_REF_INVALID,

  REFERENCE_MASTER_AXIS_REF_INVALID,
  REFERENCE_GEAR_DATA_INVALID,
  REFERENCE_GEAR_PARAMETER_INVALID,

  CHECK_DONE    := 10_000
);
END_TYPE

// ---- XTS_TRANSPORT/XtsStation/types/E_STATION_CTRL.TcDUT
{attribute 'qualified_only'}
{attribute 'strict'}
{attribute 'to_string'}
TYPE E_STATION_CTRL :
(
  STATION_CTRL_NULL,              // nothing happens here
	STATION_INIT            := 1,   // hard reset of station, list is cleared
  STATION_DISABLE         := 10,  // 
  STATION_ENABLE,                 // 

  STATION_MOVER_ENTER     := 20,  // mover may enter station
  STATION_MOVER_ENTER_RETRY,      // retry after E_STATION_STATE.STATION_ERROR_INFEED_ERROR
  STATION_MOVER_SEND,             // do not enter, send to E_STATION_STATE.STATION_MOVER_OUT

  STATION_PROCESS_START   := 30,  // double handshake with extern
  STATION_PROCESS_DONE,           // single handshake with extern
  STATION_PROCESS_NEST_SKIP,

  STATION_MOVER_OUT       := 50,  // mover may leave station now; ticket for mover is checked here (ST_STATION_CTRL.nTargetStation)
  STATION_MOVER_OUT_RETRY,        // retry after E_STATION_STATE.STATION_ERROR_OUTFEED_ERROR

  STATION_MOVER_GONE      := 60   // mover has left station, last handshake station is empty

)USINT;
END_TYPE

// ---- XTS_TRANSPORT/XtsStation/types/E_STATION_GEAR_DISTANCE_AXIS.TcDUT
{attribute 'qualified_only'}
{attribute 'strict'}
{attribute 'to_string'}
TYPE E_STATION_GEAR_DISTANCE_AXIS :
(
  // which axis nSync distance is checked for termination of GearInPosCA.
  // after nSync distance the station does a regular outfeed to target station
	FOLLOW_THE_MASTER,
  FOLLOW_THE_SLAVE
)UINT;
END_TYPE

// ---- XTS_TRANSPORT/XtsStation/types/E_STATION_STATE.TcDUT
{attribute 'qualified_only'}
{attribute 'to_string'}
TYPE E_STATION_STATE :
(
	STATION_NO_INIT,                // startup state after power on, first cycle Init of station, switches to INIT when done

  STATION_INIT,                   // CONTINUE to DISABLE
                                  // State.MoverId deleted

  STATION_DISABLE         := 10,  // + CTRL.STATION_ENABLE  --> CONTINUE to DETECT_MOVER 
                                  // station is empty, no mover is handled, check enable from ctrl

  STATION_ENABLE,                 // init of work vars, check enable from ctrl

  STATION_DETECT_MOVER,           // (QueueCount > 0)       --> CONTINUE to MOVER_ENTER

  STATION_MOVER_ENTER     := 20,  // + CTRL.MOVER_ENTER     --> CONTINUE to PROCESS_START
                                  // + CTRL.MOVER_SEND      --> CONTINUE to MOVER_OUT
                                  // mover asking for entry

  STATION_MOVER_IN_TARGET,        // (MoveToPos==TRUE)      --> CONTINUE to PROCESS_START
                                  // mover is moving to PosWait + PosStop[_nNest]

  STATION_PROCESS_START   := 30,  // + CTRL.PROCESS_START   --> CONTINUE to PROCESS_START
                                  // + CTRL.PROCESS_DONE    --> CONTINUE to CHECK
                                  // wait until process started

  STATION_PROCESS_DONE,           // + CTRL.PROCESS_DONE    --> CONTINUE to CHECK
                                  // wait until process done

  STATION_CHECK           := 40,  // check for next nest in mask, 
                                  // (mask<>0) --> CHECK_NEST
                                  // (mask==0) --> MOVER_OUT

  STATION_CHECK_NEST,             // + CTRL.MOVER_ENTER     --> CONTINUE to MOVER_IN_TARGET
                                  // get next nest position

  STATION_MOVER_OUT       := 50,  // + CTRL.MOVER_OUT       --> CONTINUE to MOVER_RELEASE
                                  // mover asking to leave

  STATION_MOVER_RELEASE,          // (MoverSendToPos==TRUE) --> CONTINUE to MOVER_GONE
                                  // mover is released + check if release distance is passed

  STATION_MOVER_WRITE_TARGET,     // worker state to write mover ticket

  STATION_MOVER_GONE      := 60,  // + CTRL.MOVER_GONE      --> CONTINUE to INIT
                                  // mover out of station, enter mover in target station list


  STATION_ERROR_NULL      := 127,
  STATION_ERROR_LIST_GET_HEAD_FAULT,    // fatal error in linked list, must never occurr, must be debugged
  STATION_ERROR_LIST_REMOVE_HEAD_FAULT, // fatal error in linked list, must never occurr, must be debugged
  STATION_ERROR_LIST_ADD_TAIL_FAULT,    // fatal error in linked list, must never occurr, must be debugged

  STATION_ERROR_LIST_STATION_ID_WRONG,  // ticket data in Queue contains wrong Station Id, can be overruled by ctrl

  STATION_ERROR_LIST_MOVER_ID_INVALID,  // fatal error in ticket data, MoverId is out of range, must be fixed by ctrl, must be debugged

  STATION_ERROR_INFEED_ERROR,           // motion error during movement, retry must be triggered by ctrl
  STATION_ERROR_OUTFEED_ERROR,          // motion error during movement, retry by ctrl OR leave by ctrl

  STATION_ERROR_OUTFEED_TARGET_INVALID, // ticket data for nTargetStation is not plausible, can be fixed by ctrl

  STATION_ERROR_FATAL     := 255 // the thing that must not be, all fatal errors end up here
)USINT;
END_TYPE

// ---- XTS_TRANSPORT/XtsStation/types/E_STATION_TYPE.TcDUT
{attribute 'qualified_only'}
{attribute 'strict'}
{attribute 'to_string'}
TYPE E_STATION_TYPE :
(
	INVALID,
  STATION_PROCESS,      // default station with/without process
  STATION_GEAR_IN_POS   // GearInPos station for flying saw with MasterAxis
)USINT;
END_TYPE

// ---- XTS_TRANSPORT/XtsStation/types/ST_STATION_CTRL.TcDUT
{attribute 'pack_mode' := '2'}
TYPE ST_STATION_CTRL :
STRUCT
  Cmd             : E_STATION_CTRL;
  {attribute 'displaymode':='bin'}
  nMask           : BYTE;           // nest mask for sending mover to next station
  nTargetStation  : USINT;          // where to next?
  rOffset         : REAL;           // optional offset for mover in target station when leaving sending station; 
                                    // use case: position correction of workpiece on wpc by vision
END_STRUCT
END_TYPE

// ---- XTS_TRANSPORT/XtsStation/types/ST_STATION_GEAR_PARAMETER.TcDUT
TYPE ST_STATION_GEAR_PARAMETER :
STRUCT
  eDistance           : E_STATION_GEAR_DISTANCE_AXIS; // follow which leader?
  rSyncDistance       : LREAL := 100.0;               // synchrone distance while the mover is geared in
  rMinDistanceToSync  : LREAL := 100.0;               // minimum distance for mover to get nSync with the Master
END_STRUCT
END_TYPE

// ---- XTS_TRANSPORT/XtsStation/types/ST_STATION_LIST_RESULT.TcDUT
TYPE ST_STATION_LIST_RESULT :
STRUCT
  wState    : WORD;   // wState == 0 --> all ok
  nIndex    : ULINT;
  stData    : ST_STATION_MOVER_DATA;  // copy of list entry
END_STRUCT
END_TYPE

// ---- XTS_TRANSPORT/XtsStation/types/ST_STATION_MOVER_DATA.TcDUT
{attribute 'pack_mode' := '2'}
TYPE ST_STATION_MOVER_DATA :
STRUCT
  nMoverId        : USINT;  // who am I?  !! MUST be correct !! - movement to base position sets everything in order, DO NOT manipulate!
  nTargetStation  : USINT;  // where shall I be? used for double checking with StationId at infeed of mover into station

  {attribute 'displaymode':='bin'}
  nMask           : BYTE;   // how many of you are there? (1 = default, no action required)

  rOffset         : REAL;   // offset for use in work flow !! added to static mover offset for every nest(bit) in nMask!!
END_STRUCT
END_TYPE

// ---- XTS_TRANSPORT/XtsStation/types/ST_STATION_PARAMETER.TcDUT
TYPE ST_STATION_PARAMETER :
STRUCT
  eType             : E_STATION_TYPE := 1;  // StationProcess or StationGearInPos
  sText             : STRING(80);           // only description
  rPosWait          : REAL;                 // start of station, 
                                            // a sending station is using this value 
                                            // to send mover to

  rReleaseDistance  : REAL;                 // distance mover has to travel (from ActPos) 
                                            // in order for station to go back to disable

  rGap              : REAL;
  rVelo             : REAL;
  rAccDec           : REAL;
  rJerk             : REAL;

  // how many nests (stop positions) mover has to stop at (1 = default)
  nConfiguredStopCount  : USINT := 1; // 1-8 --> NestMask = BYTE

  // mover stop position in station, relative to rPosWait!!
  rPosStop          : ARRAY[1..8] OF LREAL;
END_STRUCT
END_TYPE

// ---- XTS_TRANSPORT/XtsStation/types/ST_STATION_STATE.TcDUT
{attribute 'pack_mode' := '2'}
TYPE ST_STATION_STATE :
STRUCT
  State           : E_STATION_STATE;
  {attribute 'displaymode':='bin'}
  nMask           : BYTE;
  nMoverId        : USINT;
  rMoverModPos    : LREAL;            // modulo position of detected mover
  nQueue          : USINT;            // queue count for station
END_STRUCT
END_TYPE

// ---- XTS_TRANSPORT/XtsStation/types/T_NEST_OFFSET.TcDUT
TYPE T_NEST_OFFSET : ARRAY[1..MAX_MOVER]        OF
                     ARRAY[1..MAX_STATION_NEST] OF LREAL;
END_TYPE

// ---- XTS_TRANSPORT/XtsTransportUnit/types/E_XTS_TRANSPORT_CHECK.TcDUT
{attribute 'qualified_only'}
{attribute 'to_string'}
TYPE E_XTS_TRANSPORT_CHECK :
(
  // info for cyclic checks
  INIT_CHECK,
  START_CHECK,    // check cycle start
  XPU_INIT,       // Xpu: initialization


  // errors in fb_TransportUnit.Check()
  POINTER_CHECK           := 9000,
  POINTER_NULL_CTRL,

  POINTER_NULL_STATE,
  POINTER_NULL_XPU_CTRL,

  POINTER_NULL_XPU_STATE,
  POINTER_NULL_XPU_INFO,

  POINTER_NULL_GROUP_ITF,
  POINTER_NULL_GROUP_INFO,

  POINTER_NULL_MOVER,
  POINTER_NULL_MOVER_ITF,

  POINTER_NULL_MOVER_INFO,
  POINTER_NULL_MOVER_LAST_POS,
  POINTER_NULL_MOVER_LAST_GAP,

  POINTER_NULL_STATION_START,
  POINTER_NULL_STATION_ITF,
  POINTER_NULL_STATION_CONTROL,
  POINTER_NULL_STATION_STATE,
  POINTER_NULL_STATION_CTRL_ITF,

  DONE_CHECK              := 10000
)UINT;
END_TYPE

// ---- XTS_TRANSPORT/XtsTransportUnit/types/E_XTS_TRANSPORT_CTRL.TcDUT
{attribute 'strict'}
{attribute 'to_string'}
TYPE E_XTS_TRANSPORT_CTRL :
(
  CMD_NULL,
  CMD_INIT                  := 10,  // Xpu, Group, Mover initialization: clear errors, clear group, check Xpu data, check mover detection
  CMD_IDLE,

  CMD_MOVER_ENABLE          := 20,  // all mover are enabled, checked for ControlLoopClosed
  CMD_MOVER_DISABLE,                // all mover are disabled, no axis in CaGroup: no error, any axis in CaGroup: group error
  CMD_MOVER_HALT_CA,                // all movers are stopped with MC_HaltCA[]. ONLY use if all movers are in CA group
  CMD_MOVER_STOP,

  CMD_GROUP_CLEAR           := 30,  // halt all movers, clear errors, remove all movers from group, clear group
  CMD_GROUP_BUILD,                  // add all movers to group
  CMD_GROUP_ENABLE,                 // group with movers is enabled
  CMD_GROUP_STOP,                   // moving CA Group is stopped

  CMD_TRANSPORT_START       := 40,  // move all mover[i] to start position
  CMD_TRANSPORT_RESTART             // move all mover[i] to LastPosition[i]

)UINT;
END_TYPE

// ---- XTS_TRANSPORT/XtsTransportUnit/types/E_XTS_TRANSPORT_STATE.TcDUT
{attribute 'to_string'}
TYPE E_XTS_TRANSPORT_STATE :
(
  TRANSPORT_NULL,
  TRANSPORT_INVALID,
  TRANSPORT_INIT            := 10,  // Xpu, Group, Mover initialization: init TcCOM objects, clear errors, clear group, check Xpu data, check mover detection
  TRANSPORT_IDLE,                   // cyclic check for errors, check Xpu data

  TRANSPORT_MOVER_ENABLE    := 20,  // all mover are enabled, checked for ControlLoopClosed
  TRANSPORT_MOVER_DISABLE,          // all mover are disabled
  TRANSPORT_MOVER_HALT_CA,          // all mover standstill
  TRANSPORT_MOVER_STOP,

  TRANSPORT_GROUP_CLEAR     := 30,  // halt all movers, clear errors, remove all movers from group, clear group
  TRANSPORT_GROUP_BUILD,            // add all movers to group
  TRANSPORT_GROUP_ENABLE,           // group with movers is enabled
  TRANSPORT_GROUP_STOP,             // CaGroup Stop, CaGroup Reset, All movers halt

  TRANSPORT_START           := 40,  // move all mover[i] to start position
  TRANSPORT_RESTART                 // move all mover[i] to LastPosition[i]
)UINT;
END_TYPE

// ---- XTS_TRANSPORT/XtsTransportUnit/types/ST_XTS_TRANSPORT_CTRL.TcDUT
{attribute 'pack_mode' := '2'}
TYPE ST_XTS_TRANSPORT_CTRL :
STRUCT
  Cmd       : E_XTS_TRANSPORT_CTRL;
END_STRUCT
END_TYPE

// ---- XTS_TRANSPORT/XtsTransportUnit/types/ST_XTS_TRANSPORT_STATE.TcDUT
{attribute 'pack_mode' := '2'}
TYPE ST_XTS_TRANSPORT_STATE :
STRUCT
  State         : E_XTS_TRANSPORT_STATE;  // combined value of state and result(e_progress); (hint: extract state value by mod division)
  Check         : E_XTS_TRANSPORT_CHECK;

  XpuState      : ST_XPU_STATE;
  XpuInfo       : ST_XPU_INFO;
  GroupInfo     : ST_GROUP_INFO; 
END_STRUCT
END_TYPE

// ---- XTS_TRANSPORT/_Visualization/types/ST_XPU_STRINGS.TcDUT
TYPE ST_XPU_STRINGS :
STRUCT
  sXpuState       ,
  sXpuResult      ,
  sXpuCyclicCheck ,
  sXpuOpMode      ,
  sXpuMoverId_DetectionMode,
  sXpuMoverPosAssignement : STRING(30) := 'NULL';
END_STRUCT
END_TYPE

// ---- _MSG/types/e_Device.TcDUT
{attribute 'to_string'}
TYPE e_Device :
(
  Device_Null,                  // NULL               - not to be used
  Device_Main,                  // MAIN(PRG)          - reserved for MAIN(PRG)
  Device_MainAxis,              // MAIN_AXIS(PRG)     - reserved for MAIN_AXIS(PRG)
  Device_Nci,                   // NCI(PRG)           - reserved for NCI(PRG)
  Device_Cam,                   // CAM(PRG            - reserved for CAM(PRG)
  Device_Functions,             // FUNCTIONS(PRG)     - reserved for FUNCTIONS(PRG)
  Device_FlyingSaw,             // FLYING_SAW(PRG)    - reserved for FLYING_SAW(PRG)
  Device_MainApplication,       // MAIN_APP(PRG)      - reserved for MAIN_APP(PRG)

  Device_MoverSelector,         // single mover interface for xts applications
  Device_ParameterSelector,     // fb_ParameterSelector can only exist once in a project.
  Device_Configuration,         // fb_Configuration can handle multiple files therefore only one instance is required
  Device_XmlData,               // generic XML Data (e.g. persistent data)
  Device_Utilities,             // service calls to anyone you may want to talk to, the main intent is to get XPU and TcXtsIo data to the application side

  General           :=  1000,
  CaGroup           :=  2000,
  Xpu               :=  3000,
  XpuCtrl           :=  4000,
  Mover             :=  5000,
  MoverCtrl         :=  6000,
  XtsTransportUnit  :=  7000,
  XfcTriggerBox     :=  8000,
  XfcTouchProbe     :=  9000,
  XtsStation        := 10000,

  Camming           := 11000,
  NciChannel        := 12000,
  NciChannelCtrl    := 13000,
  Axis              := 14000,
  XfcAxis           := 15000,

  // txt file logging LOG_FILE_METRICS
  MetricsXts        := 16000,   //entries from xts Metrics are written into dedicated txt file (see f_MessageSet, here's the diverter)
  MetricsAxis       := 17000,   //entries from PLC_MOTION Metrics are written into dedicated txt file

  // txt file logging LOG_FILE_APP
  Process           := 20000,   // entries from process are written into dedicated txt file.
  ProcessListCtrl   := 21000,
  TicketListCtrl    := 22000,

  Application       := 30000,   // entries from application are written into dedicated txt file.


  // txt file logging LOG_FILE_PRODUCT - this is for you to use
  DataProduct       := 40000
)UDINT;
END_TYPE

// ---- _MSG/types/E_MessageType.TcDUT
{attribute 'strict'}
{attribute 'to_string'}
TYPE E_MessageType :
(
  //-----------------------------------------------------
  //-----------------------------------------------------
  //  message system:
  //  - errors are always calling f_MessageSet()
  //  - errors are always entered into its list
  //
  //  - message severity is set by this enum (like everywhere else)
  //
  //  - message frequency is set by this enum
  //    - IF you get above 50 stations, 
  //      writing to the file system takes time:
  //
  //    Batch: switching on metrics (> Empty) must not add cpu load, 
  //      --> so do not clutter here
  //
  //    Info:  regular flow of information (>Error / >Warning) 
  //           must not add significant cpu load, 
  //      --> so do not clutter here
  //
  //    Verbose and above:
  //    --> for small systems (< 96 mover, < 50 stations) 
  //        you may switch it on for everybody, 
  //        files get big quickly ;-)
  //
  //    --> switch on during test phase for a handful of stations
  //
  //    --> high detail logging always and for everybody
  //    --> we need somebody who transfers data more quickly
  //      --> I can offer a .NET(C#) ADS tool which collects the list.
  //          .NET application then pushes to database
  //-----------------------------------------------------
  //-----------------------------------------------------
  eMessageEmpty,    // he who is without bounds may speak
  eMessageBatch,    // he who counts words, counts numbers (Batch started, Next in Batch, Batch done)
  eMessageError,    // mine, your(')s, anybody's, let the numbers tell you
  eMessageWarning,  // I told you so
  eMessageInfo,     // A long time ago in a galaxy far, far away...
  eMessageVerbose,  // He talks a lot, doesn't he?; Yeah! He's very knowledgeable.
  eMessageSentient  // Keep them out of bright light, Don't get them wet, do not feed them after midnight!! No matter how much they beg!!
)DINT;
END_TYPE

// ---- _MSG/types/E_MESSAGE_BATCH.TcDUT
{attribute 'qualified_only'}
{attribute 'strict'}
{attribute 'to_string'}
TYPE E_MESSAGE_BATCH :
(
	MSG_BATCH_NULL,
  MSG_BATCH_JOB_STARTED,
  MSG_BATCH_NEXT_IN_JOB,
  MSG_BATCH_JOB_DONE
)UINT;
END_TYPE

// ---- _MSG/types/E_MESSAGE_CHECK.TcDUT
{attribute 'qualified_only'}
{attribute 'strict'}
{attribute 'to_string'}
TYPE E_MESSAGE_CHECK :
(
  NULL,
  // 9000 --> here comes your error
  POINTER_INVALID             := 9000,
  POINTER_TIME_INVALID,
  POINTER_LIST_INVALID,
  POINTER_MSG_IDX_INVALID,
  POINTER_ERR_IDX_INVALID,
  POINTER_ROOT_FILE_INVALID,
  POINTER_ROOT_DIR_INVALID,
  POINTER_CTRL_INVALID,
  POINTER_STATE_INVALID,

  // 10000 --> here comes your man
  CHECK_DONE                        := 10000
)UINT;
END_TYPE

// ---- _MSG/types/E_MESSAGE_CTRL.TcDUT
{attribute 'qualified_only'}
{attribute 'strict'}
{attribute 'to_string'}
TYPE E_MESSAGE_CTRL :
(
	MSG_CTRL_NULL,
	MSG_CTRL_INIT   := 10,
  MSG_CTRL_IDLE   := 30,
  MSG_CTRL_WRITE  := 50
)UINT;
END_TYPE

// ---- _MSG/types/E_MESSAGE_FLOW.TcDUT
{attribute 'qualified_only'}
{attribute 'strict'}
{attribute 'to_string'}
TYPE E_MESSAGE_FLOW :
(
  MSG_FLOW_INIT,
  MSG_FLOW_ROOT                 := 10,
  MSG_FLOW_ROOT_CREATE,
  MSG_FLOW_ROOT_CREATE_BUSY,
  MSG_FLOW_FOLDER,
  MSG_FLOW_FOLDER_CREATE,
  MSG_FLOW_FOLDER_CREATE_BUSY,
  MSG_FLOW_FILE_CREATE_DONE,
  MSG_FLOW_LINE_START           := 100,
  MSG_FLOW_LINE_BUILD,
  MSG_FLOW_LINE_CHECK,
  MSG_FLOW_WRITE_FILE_BUSY      := 200,
  MSG_FLOW_WRITE_FILE_END,
  MSG_FLOW_WRITE_FILE_DONE      := 1000
)UINT;
END_TYPE

// ---- _MSG/types/E_MESSAGE_STATE.TcDUT
{attribute 'qualified_only'}
//{attribute 'strict'}
{attribute 'to_string'}
TYPE E_MESSAGE_STATE :
(
	MSG_STATE_NULL,
  MSG_STATE_INIT    := 10,
  MSG_STATE_IDLE    := 30,
  MSG_STATE_WRITE   := 50
)UINT;
END_TYPE

// ---- _MSG/types/e_Subdevice.TcDUT
{attribute 'strict'}
{attribute 'to_string'}
TYPE e_Subdevice :
(
  // sub device for message system
  General                 :=  0,
  MainInit,
  // Motion Control FB Instances
  fbPower,
  fbReset,
  fbResetSercos,
  fbHalt,
  fbStop,                 // 5
  fbHome,
  fbJog,
  fbMoveVelocity1,
  fbMoveVelocity2,
  fbMoveAbsolute1,        // 10
  fbMoveAbsolute2,
  fbMoveEndless,
  fbMovePtP,
  fbMoveVelo,
  fbSendToPos,

  // CA CollisionAvoidance FB instances
  // CA group fb instances
  fbCaGroup             := 30,
  fbMoveToPosCa,
  fbSendToAbsPosCa,
  fbSendToModuloPosCa,
  fbGearInPosCa,
  fbGroupAddAxis,
  fbGroupRemoveAxis,
  fbGroupDisable,
  fbGroupEnable,
  fbGroupErrorRead,
  fbGroupStatusRead,
  fbGroupReset,
  fbGroupStop,
  fbHaltCa,

  fbGearIn                := 50,
  fbGearOut,
  fbGearInMultiMaster,

  fbCamOutV2              := 80,
  fbCamInV2,
  fbCamScalingV2,
  fbCamInfoV2,
  fbReadMotionFunction,
  fbReadMotionFunctionPoint,
  fbReadMotionFunctionValues,
  fbWriteMotionFunction,
  fbWriteMotionFunctionPoint,
  fbSetOnlineChangeMode,

  fbReadParameter         := 100,
  fbReadBoolParameter,
  fbWriteParameter,
  fbWriteBoolParameter,
  fbWriteParameterPersistent,
  fbXmlRead,
  fbXmlWrite,
  fbCreateFolder,

  fbBuildGroup            := 200,
  fbClearGroup,
  fbLoadProg,
  fbResetItp,
  fbStartStopItp,
  fbEStopItp,             // 205
  fbStepOnAfterEStopItp,
  fbConfirmHskItp,
  fbDelDtgItp,
  fbNciFeedTablePreparation,
  fbNciFeedTable,         // 210
  fbReadLine,
  fbItpReadRParams,
  fbItpWriteRParams,
  Get_ItpState,
  Get_Error,              // 215


  XfcPositionAtTime       := 300,
  XfcTimeOfPosition,
  XfcTimeToPosition,
  XfcTimeToModuloPosition,
  XfcRecordedPosition,
  XfcTouchProbe,          // 305
  XfcTouchProbeEL1258,
  XfcTouchProbeOptions,
  XfcTriggerRef,
  XfcTriggerRef_MT,
  XfcEl1258Interface_MT,  // 310
  XfcRecordedPosition_MT,
  XfcTriggerOut,
  XfcTriggerStart,
  XfcSwitchOn_2252,
  XfcSwitchOff_2252,      // 315
  XfcInit,
  XfcLatchPosition,
  XfcWaitForPosition,

  AxisMode              := 1000,
  AxisControl,
  AxisStartUp,
  AxisCycle,
  AxisIdle,

  NciControl            := 2000,
  NciStartUp,
  NciCycle,
  NciIdle,

  FlyingSawControl      := 2100,
  FlyingSawStartUp,

  StationLinkedList     := 3000,
  StationInitList,
  StationAddHead,
  StationAddTail,
  StationGetHead,
  StationRemoveHeadValue,
  StationGearInDistanceToSync,
  StationGearInSyncStart,
  StationGearInSyncMove,
  StationGearInSyncEnd,
  StationCalcInfeedPosition,

  StationControl        := 4000,
  StationState, 

  Xpu_fbEnvironment     := 5000,
  Xpu_fbProcessingUnit,
  Xpu_fbXpuPart,
  Xpu_fbXpuTrack,
  Xpu_fbMc2CaGroup,
  Xpu_fbParameterSet,
  Xpu_fbNctController,

  Xpu_fbPartModules     := 5500,

  Xpu_fbMoverXpu        := 6000,

  Xpu_fbNctBaseUnit     := 6500,

  TransportUnit_General := 7000,
  TransportUnit_Restart := 7010,
  TransportUnit_Start,
  TransportUnit_XpuInit,
  TransportUnit_StationClearOutfeed,
  TransportUnit_GroupEnable,
  TransportUnit_GroupClear,
  TransportUnit_GroupBuild,
  TransportUnit_GroupStop,
  TransportUnit_MoverEnableAll,
  TransportUnit_MoverDisableAll,


  CamControl            := 8000,
  CamStartUp,
  CamCycle,

  Process_StationCollector    := 11000,
  Process_ProcessCollector    := 11100,
  Process_ProcessCollector_Init,
  Process_ProcessCollector_Cycle,
  Process_ProcessCollector_Control,

  Process_LinkedList_GetHead,
  Process_LinkedList_RemoveHead,
  Process_LinkedList_AddTail,
  Process_LinkedList_CheckData,
  Process_StationQueue_Check,

  Process_LinkedList_Com              := 11200,
  Process_LinkedList_Com_Init,
  Process_LinkedList_Com_Cmd,
  Process_LinkedList_Com_AddHead,
  Process_LinkedList_Com_AddTail,
  Process_LinkedList_Com_DelHead,
  Process_LinkedList_Com_DelTail,
  Process_LinkedList_Com_GetHead,
  Process_LinkedList_Com_GetTail,


  Instance_Command              := 12000,
  Instance_ProcessConductor,
  Instance_BufferInfeed,
  Instance_Infeed,
  Instance_BufferOutfeed,
  Instance_Outfeed,
  Instance_Sender_Buffer,

  Ticket_LinkedList_Ctrl        := 12100,
  Ticket_LinkedList_Com_Init,
  Ticket_LinkedList_Com_Cmd,
  Ticket_LinkedList_Com_AddHead,
  Ticket_LinkedList_Com_AddTail,
  Ticket_LinkedList_Com_DelHead,
  Ticket_LinkedList_Com_DelTail,
  Ticket_LinkedList_Com_GetHead,
  Ticket_LinkedList_Com_GetTail,
  

  Application                 := 13000,
  Application_Check,
  Application_Clear,
  Application_Cmd,
  Application_Disable,
  Application_Enable,
  Application_Finish,
  Application_Init,
  Application_Proceed,
  Application_Work,

  Utilities                   := 13100,
  Utilities_GetStationOnModule,
  Utilities_SetGlobalConstraints

)DINT;
END_TYPE

// ---- _MSG/types/ST_Message.TcDUT
TYPE ST_Message :
STRUCT
  eType         : e_MessageType;
  eDevice       : e_Device;
  eSubdevice    : e_SubDevice;
  {attribute 'displaymode':='hex'}
  iErrorNumber  : LINT;
  tTime         : STRING(24);
  sText         : STRING(127);
END_STRUCT
END_TYPE

// ---- _MSG/types/ST_MESSAGE_CTRL.TcDUT
TYPE ST_MESSAGE_CTRL :
STRUCT
  Cmd         : E_MESSAGE_CTRL;
END_STRUCT
END_TYPE

// ---- _MSG/types/ST_MESSAGE_STATE.TcDUT
TYPE ST_MESSAGE_STATE :
STRUCT
  State         : E_MESSAGE_STATE;  // as always... combined value of Cmd equivalent and e_progress
END_STRUCT
END_TYPE

// ---- _XML/Configuration/types/ST_Configuration.TcDUT
TYPE ST_Configuration :
STRUCT
  XtsStationParameter  : ARRAY[1..MAX_STATION] OF ST_STATION_PARAMETER;
END_STRUCT
END_TYPE

// ---- _XML/PositionOffsets/types/ST_MOVER_OFFSETS.TcDUT
TYPE ST_MOVER_OFFSETS :
STRUCT
  // static position offsets in stations
  PositionOffset      : ARRAY[1..MAX_STATION] OF T_NEST_OFFSET; // added to PosStop[] in XtsStation
END_STRUCT
END_TYPE

// ---- _XML/types/E_DATA_CHECK.TcDUT
{attribute 'qualified_only'}
{attribute 'strict'}
{attribute 'to_string'}
TYPE E_DATA_CHECK :
(
  NULL,
  REFERENCE_CTRL_INVALID  := 9000,
  REFERENCE_STATE_INVALID,

  POINTER_STATION_PARAMETER_INVALID := 9100,
  POINTER_MOVER_DISTANCES_INVALID,
  POINTER_MOVER_OFFSETS_INVALID,

  DONE_CHECK              := 10000
);
END_TYPE

// ---- _XML/types/E_DATA_CTRL.TcDUT
{attribute 'qualified_only'}
{attribute 'to_string'}
{attribute 'strict'}
TYPE E_DATA_CTRL :
(
  NULL,
	INIT  := 10,
  READ  := 20,
  WRITE := 30
)UINT;
END_TYPE

// ---- _XML/types/E_DATA_STATE.TcDUT
{attribute 'qualified_only'}
{attribute 'to_string'}
TYPE E_DATA_STATE :
(
	NULL,
  NO_EXIST,
  INIT        := 10,
  READ        := 20,
  WRITE       := 30
)UINT;
END_TYPE

// ---- _XML/types/ST_DATA_CTRL.TcDUT
{attribute 'pack_mode' := '2'}
TYPE ST_DATA_CTRL :
STRUCT
  Cmd       : E_DATA_CTRL;
END_STRUCT
END_TYPE

// ---- _XML/types/ST_DATA_STATE.TcDUT
{attribute 'pack_mode' := '2'}
TYPE ST_DATA_STATE :
STRUCT
  State       : E_DATA_STATE;
  Init        : E_PROGRESS;
END_STRUCT
END_TYPE

// ---- PLC_MOTION/_GVL/PLC_CONSTANT.TcGVL
//{attribute 'qualified_only'}
VAR_GLOBAL CONSTANT


  //-----------------------------------------------------------------------------
  // AXIS related limits
  //-----------------------------------------------------------------------------
  MAX_AXIS              : UINT    := 3;
  MAX_RETRY             : UINT    := 5;


  //-----------------------------------------------------------------------------
  // NCI related limits and *.nc standard folder
  //-----------------------------------------------------------------------------
{IF NOT defined (BSD)}
  NCI_DIR               : STRING  := 'C:\TwinCAT\Mc\Nci\';
{ELSE}
  NCI_DIR               : STRING  := '/usr/local/etc/TwinCAT/Mc/Nci/';
{END_IF}

{IF defined (NCI)}
  {info 'PLC_MOTION_LAYER: NCI'}
  NCI_ACTIVE            : BOOL    := TRUE;
  CONFIG_NAME           : STRING  := 'NCI_Spec_Ch_';
{ELSE}
  NCI_ACTIVE            : BOOL    := FALSE;
  CONFIG_NAME           : STRING  := 'NCI_NOT_ACTIVE';
{END_IF}

  MAX_NCI_CH            : UINT    := 1;

  MAX_PATH_STEPS        : UINT    := 5;
  MAX_MC_AXIS           : UINT    := 3;
  MAX_AUX_AXIS          : UINT    := 2;
  MAX_R_PARA            : UINT    := 10;


  //-----------------------------------------------------------------------------
  // CAMMING related limits
  //-----------------------------------------------------------------------------
{IF defined (CAM)}
  {info 'PLC_MOTION_LAYER: CAM'}
  CAM_ACTIVE                  : BOOL    := TRUE;
{ELSE}
  CAM_ACTIVE                  : BOOL    := FALSE;
{END_IF}

  MAX_CAM_CH                  : UINT    := 1;

  MAX_MOTION_FUNCTION_POINTS  : UINT    := 10;

  // HAUD
  // 17.07.2024
  // Start Implementation of Position Trigger function
  //  - Timestamp/position output
  //  - Latch DC time from input
  
  MAX_TRIGGER_BOX             : UINT := 12;
  MAX_TOUCH_PROBE             : UINT := 12;
  MAX_TRIGGER_COUNT           : UINT :=  4;
  MAX_MTI_CH                  : UINT :=  1; // MAX mti channel per EL terminal

{IF defined (XFC)}
  {info 'PLC_MOTION_LAYER: XFC'}
  XFC_ACTIVE                  : BOOL := TRUE;
{ELSE}
  XFC_ACTIVE                  : BOOL := FALSE;
{END_IF}

  // HAUD
  // 2026 05 28
  // Gear In Pos implementation for flying saw application 

{IF defined (SAW)}
  {info 'PLC_MOTION_LAYER: FLYING_SAW'}
  FLY_SAW_ACTIVE              : BOOL  := TRUE;
{ELSE}
  FLY_SAW_ACTIVE              : BOOL  := FALSE;
{END_IF}
END_VAR

// ---- XTS_TRANSPORT/GVL_XTS_CONSTANTS.TcGVL
//{attribute 'qualified_only'}
VAR_GLOBAL CONSTANT
//-----------------------------------------------------------------------------------------------------------------------------------------
//-----------------------------------------------------------------------------------------------------------------------------------------
//
//  HAUD 2026.03.15
//  - parameter list deleted (never used the parameter feature anyway), 
//    back to static global constants
//
//-----------------------------------------------------------------------------------------------------------------------------------------
//-----------------------------------------------------------------------------------------------------------------------------------------
//  Connections to XTS Utility Lib data: 
//  - suits this simple approach, 
//  - leaves you options to expand, 
//  - expansion and multiplication is not implemented here on purpose, 
//  - this project is designed to get the main ideas across, 
//  - setting up a matrix for multiple fb_Xpu instances with it, 
//    --> a second step you might want to organize from here; 
//        --> I leave the details up to you
//-----------------------------------------------------------------------------------------------------------------------------------------
//-----------------------------------------------------------------------------------------------------------------------------------------
  MAX_MOVER           : UINT    := TO_UINT(Tc3_XTS_Utility.TcIoXtsEnvironmentParameterList.MaxXtsMoversPerXpu);
  MAX_MODULE          : UINT    := TO_UINT(Tc3_XTS_Utility.TcIoXtsEnvironmentParameterList.MaxModulesPerPart);
  MAX_PART            : UINT    := TO_UINT(Tc3_XTS_Utility.TcIoXtsEnvironmentParameterList.MaxXtsPartsPerXpu);
  MAX_TRACK           : UINT    := TO_UINT(Tc3_XTS_Utility.TcIoXtsEnvironmentParameterList.MaxXtsTracksPerXpu);
  MAX_GROUP           : UINT    := TO_UINT(Tc3_XTS_Utility.TcIoXtsEnvironmentParameterList.MaxXtsCaGroup);

  MAX_INFO_SERVER     : UINT    := TO_UINT(Tc3_XTS_Utility.TcIoXtsEnvironmentParameterList.MaxXtsInfoServer);
  MAX_INFO_STATION    : UINT    := TO_UINT(Tc3_XTS_Utility.TcIoXtsEnvironmentParameterList.MaxXtsInfoStation);
  MAX_INFO_STOP_POS   : UINT    := TO_UINT(Tc3_XTS_Utility.TcIoXtsEnvironmentParameterList.MaxXtsStopPositionsPerStation);

  MAX_PARAMETER_SET   : UINT    := TO_UINT(Tc3_XTS_Utility.TcIoXtsEnvironmentParameterList.MaxXtsParameterSet);

  MAX_NCT_BASE_UNIT   : UINT    := TO_UINT(Tc3_XTS_Utility.TcIoXtsEnvironmentParameterList.MaxXtsNctBaseUnitInterfaces);
//-----------------------------------------------------------------------------------------------------------------------------------------
//-----------------------------------------------------------------------------------------------------------------------------------------
//  XTS_TRANSPORT_LAYER
//  - project constants you will have to adjust in order to build your transport logic
//-----------------------------------------------------------------------------------------------------------------------------------------
//-----------------------------------------------------------------------------------------------------------------------------------------
  MAX_STATION         : UINT    := 21;

  MAX_STATION_NEST    : UINT    := TO_UINT(SIZEOF(ST_STATION_STATE.nMask)*8);
  MAX_LIST_NODES      : UINT    := MAX_MOVER;
  MAX_MASTER          : UINT    := 1;
//-----------------------------------------------------------------------------------------------------------------------------------------
//-----------------------------------------------------------------------------------------------------------------------------------------
END_VAR

// ---- _MSG/GVL_MSG_XTS.TcGVL
{attribute 'qualified_only'}
VAR_GLOBAL CONSTANT
  //-----------------------------------------------------------------------------
  // file paths for message system
  //  - compiler define option WIN switches to Windows file paths
  //-----------------------------------------------------------------------------
{IF defined (WIN)}
  {info 'WIN folders'}
  LOG_DIR               : STRING  := 'C:\TwinCAT\#MsgFiles\';       // delimiter at the end is mandatory!!
  CON_DIR               : STRING  := 'C:\TwinCAT\#Configuration\';  // delimiter at the end is mandatory!!
{ELSE}
  {info 'BSD folders'}
  LOG_DIR               : STRING  := '/usr/local/etc/TwinCAT/#MsgFiles/';       // delimiter at the end is mandatory!!
  CON_DIR               : STRING  := '/usr/local/etc/TwinCAT/#Configuration/';  // delimiter at the end is mandatory!!
{END_IF}

  LOG_FILE              : STRING  := 'MSG_XtsTransport_';
  LOG_FILE_APP          : STRING  := 'MSG_Application_';
  LOG_FILE_METRIC       : STRING  := 'MSG_XtsTransportMetrics_';

  MAX_MESSAGE           : UINT    := 2000; // max entry in message list
END_VAR
VAR_GLOBAL
  //-----------------------------------------------------------------------------
  // Message System
  //  - Everybody uses f_MessageSet(ST_Message)
  //    - DECISION WHICH LIST IS MADE IN f_MessageSet !!
  //    - which list to use is determined by e_Device in your message
  //
  //  - MessageData instances are self sufficient and need only 
  //    datafield assignment for correct data-flow
  //
  //
  //-----------------------------------------------------------------------------
  //-----------------------------------------------------------------------------
  //-----------------------------------------------------------------------------
  // (ST_Message.eDevice := e_Device.Application)
  //----------------------------------------------------------------------------- 
  ApplicationMessageData          : fb_MessageDataCtrl;
  ApplicationMessageCtrl          : st_message_ctrl;
  ApplicationMessageState         : st_message_state;

  ApplicationMessages             : ARRAY[1..MAX_MESSAGE] OF ST_Message;
  MessageApplicationIndex         : UINT := 0; // message index for higher layers (grouping, Instances, etc.)
  MessageApplicationError         : UINT := 0; // error counter for higher learning
  //-----------------------------------------------------------------------------
  //-----------------------------------------------------------------------------
  // (ST_Message.eDevice := from Device_Null to XfcAxis)
  //-----------------------------------------------------------------------------
  TransportMessageData            : fb_MessageDataCtrl;
  TransportMessageCtrl            : st_message_ctrl;
  TransportMessageState           : st_message_state;

  TransportMessages               : ARRAY[1..MAX_MESSAGE] OF ST_Message;
  MessageTransportIndex           : UINT := 0; // message index for base layer
  MessageTransportError           : UINT := 0; // error counter for base layer
  //-----------------------------------------------------------------------------
  //-----------------------------------------------------------------------------
  // (ST_Message.eDevice := e_Device.Metrics)
  //-----------------------------------------------------------------------------
  MetricsMessageData              : fb_MessageDataCtrl;
  MetricsMessageCtrl              : st_message_ctrl;
  MetricsMessageState             : st_message_state;

  MetricsMessages                 : ARRAY[1..MAX_MESSAGE] OF ST_Message;
  MessageMetricsIndex             : UINT := 0; // message index for metrics data
  MessageMetricsError             : UINT := 0; // error counter for metrics data
  //-----------------------------------------------------------------------------
  //-----------------------------------------------------------------------------
  // (ST_Message.eDevice := e_Device.ProductData)
  //-----------------------------------------------------------------------------
  ProductMessageData              : fb_MessageDataCtrl;   // This is for you
  ProductMessageCtrl              : st_message_ctrl;
  ProductMessageState             : st_message_state;

  ProductMessages                 : ARRAY[1..MAX_MESSAGE] OF ST_Message;
  MessageProductIndex             : UINT := 0; // message index for your product data
  MessageProductError             : UINT := 0; // error counter for your product data
  //-----------------------------------------------------------------------------
  //-----------------------------------------------------------------------------
  fbLocalTime                     : fb_LocalTime;
  dtLocalTime                     : DT;
  sLocalTime                      : STRING;
  //-----------------------------------------------------------------------------
  //-----------------------------------------------------------------------------
  //-----------------------------------------------------------------------------
  //-----------------------------------------------------------------------------
  MessageLevelXpu                 : E_MessageType;
  MessageLevelStations            : ARRAY[1..MAX_STATION] OF E_MessageType;
  MessageLevelMovers              : ARRAY[1..MAX_MOVER]   OF E_MessageType;

  MessageLevelProcess             : ARRAY[1..MAX_PROCESS] OF E_MessageType;

{IF defined (TEST)}
  {info 'TEST logging enabled'}
  MessageLevel                    : E_MessageType := eMessageinfo; // a lot of messages
{ELSE}
  MessageLevel                    : E_MessageType := eMessageEmpty; // only errors are written into list 
{END_IF}

END_VAR

// ---- _MSG/I_MessageData.TcIO
INTERFACE I_MessageData

PROPERTY DirRoot : POINTER to string(255)
SET
END_SET
END_PROPERTY

PROPERTY ErrorIndex : reference to uint
SET
END_SET
END_PROPERTY

PROPERTY FileRoot : pointer to string(255)
SET
END_SET
END_PROPERTY

PROPERTY LocalTime : pointer to DT
SET
END_SET
END_PROPERTY

PROPERTY MessageIndex : reference to uint
SET
END_SET
END_PROPERTY

PROPERTY MsgList : pointer to ARRAY[1..GVL_MSG_XTS.MAX_MESSAGE] OF st_message
SET
END_SET
END_PROPERTY

END_INTERFACE

// ---- _MSG/class/fb_MessageDataCtrl.TcPOU
FUNCTION_BLOCK fb_MessageDataCtrl EXTENDS fb_MessageData
VAR
  _stCtrl       : REFERENCE TO ST_MESSAGE_CTRL;
  _stState      : REFERENCE TO ST_MESSAGE_STATE;

  _eCmd,
  _eCmdOld      : E_MESSAGE_CTRL;

  _eResult,
  _eJobResult   : E_PROGRESS;

  _eState       : E_MESSAGE_STATE;

END_VAR

//-----------------------------------------------------------------------------
// check pointers
//-----------------------------------------------------------------------------
IF NOT Check()
THEN
  _eResult                      := E_PROGRESS.PROGRESS_ERROR;
  RETURN;
END_IF
//-----------------------------------------------------------------------------
// check date
// new message file for a new day
//-----------------------------------------------------------------------------
IF (FolderDate(_dtLocalTime) <> _sFolderDate)
THEN
  _bFileCreated                 := FALSE;
END_IF
//-----------------------------------------------------------------------------
//----------------------------------------------------------------------------- 
// copy to local for debug
_eCmd                         := _stCtrl.Cmd;

// cyclic check for command change
// get state for cmd
IF (_eCmd <> _eCmdOld)
THEN
  // get matching sdtate for Ctrl.Cmd
  _eState                     := Cmd(_eCmd);
  _eCmdOld                    := _eCmd;
END_IF


CASE _eResult
OF
  E_PROGRESS.PROGRESS_INVALID:
    _stState.State            := E_MESSAGE_STATE.MSG_STATE_NULL;

  E_PROGRESS.PROGRESS_ERROR:
    _stState.State            := _eState + E_PROGRESS.PROGRESS_ERROR;

  E_PROGRESS.PROGRESS_DONE:
    _stState.State            := _eState + E_PROGRESS.PROGRESS_DONE;

ELSE
  // work in progress
  // update progress for extern use
  _stState.State              := _eState + _eResult;

  CASE _eState
  OF
    E_MESSAGE_STATE.MSG_STATE_INIT:
      _eResult                := BuildFolder(TRUE);


    E_MESSAGE_STATE.MSG_STATE_IDLE:
      IF (_nMsgIndex < GVL_MSG_XTS.MAX_MESSAGE - GVL_MSG_XTS.MAX_MESSAGE/10)
      THEN
        _eResult              := E_PROGRESS.PROGRESS_WORKING;
      ELSE
        _eResult              := E_PROGRESS.PROGRESS_DONE;
        _nMsgIndex            := 0;
        // copy from attached list to local
        memcpy(ADR(_aWriteList), _pMsgList, SIZEOF(_aWriteList));
        // clear attached list
        memset(_pMsgList, 0, SIZEOF(_aWriteList));
      END_IF


    E_MESSAGE_STATE.MSG_STATE_WRITE:
      _eResult                := BuildFileData(TRUE);

  ELSE
      _eResult               := E_PROGRESS.PROGRESS_INVALID;
  END_CASE
END_CASE

METHOD BuildFileData : e_progress
VAR_INPUT
  Execute     : BOOL;
END_VAR
VAR_INST
  _nErrorId   : UDINT;
  _eState,
  _eRes       : E_PROGRESS;
  _eFlow      : E_MESSAGE_FLOW;

  _nStringLength  : UINT;
END_VAR
//-----------------------------------------------------------------------------
IF NOT Execute 
THEN
  _eRes                           := WriteData(FALSE);
  _eRes                           := BuildFolder(FALSE);
	_eState                         := E_PROGRESS.PROGRESS_INIT; 
END_IF 
//-----------------------------------------------------------------------------
IF NOT Check() 
THEN 
	BuildFileData                   := E_PROGRESS.PROGRESS_ERROR; 
	RETURN; 
END_IF
//-----------------------------------------------------------------------------
//-----------------------------------------------------------------------------
CASE _eState
OF
  E_PROGRESS.PROGRESS_INIT:
    IF Execute
    THEN
      _nErrorId                   := 0;
      _iStart 	                  := 1;
      _iEnd 		                  := SEL((_nMsgIndex > GVL_MSG_XTS.MAX_MESSAGE-1),
                                          _nMsgIndex,
                                          GVL_MSG_XTS.MAX_MESSAGE);

      memset(ADR(_sWriteData),0,SIZEOF(_sWriteData));

      IF (_sFolderDate <> FolderDate(_dtLocalTime))
      THEN
        _eState                   := E_PROGRESS.PROGRESS_PREPARE;
      ELSE
        _eState                   := E_PROGRESS.PROGRESS_BUSY;
        _eFlow                    := E_MESSAGE_FLOW.MSG_FLOW_LINE_START;
      END_IF
    END_IF
END_CASE
//-----------------------------------------------------------------------------
//-----------------------------------------------------------------------------
CASE _eState
OF
  E_PROGRESS.PROGRESS_PREPARE:
    _eRes                         := BuildFolder(TRUE);
    CASE _eRes
    OF
      E_PROGRESS.PROGRESS_DONE:
      _eState                     := E_PROGRESS.PROGRESS_BUSY;
      _eFlow                      := E_MESSAGE_FLOW.MSG_FLOW_LINE_START;

      E_PROGRESS.PROGRESS_ERROR:
      _eState                     := E_PROGRESS.PROGRESS_ERROR;
    END_CASE
END_CASE
//-----------------------------------------------------------------------------
//-----------------------------------------------------------------------------
CASE _eState
OF
  E_PROGRESS.PROGRESS_BUSY:
  CASE _eFlow
  OF
    E_MESSAGE_FLOW.MSG_FLOW_LINE_START:
      _eRes                       := BuildFolder(FALSE);
      _nErrIndex                  := 0; // rise and shine, all quarrels erased but not forgotten
      _nMsgIndex                  := 0;
  
      // copy from attached list to local
      memcpy(ADR(_aWriteList), _pMsgList, SIZEOF(_aWriteList));
  
      // clear attached list
      memset(_pMsgList, 0, SIZEOF(_aWriteList));


      _eFlow                      := E_MESSAGE_FLOW.MSG_FLOW_LINE_BUILD;
      _iCount                     := _iStart;
  END_CASE
  CASE _eFlow
  OF
    E_MESSAGE_FLOW.MSG_FLOW_LINE_BUILD:
      _eFlow                      := E_MESSAGE_FLOW.MSG_FLOW_LINE_CHECK;
      IF (_aWriteList[_iCount].eType > E_MessageType.eMessageEmpty)
      THEN
        _sTmp                     := TO_STRING(_aWriteList[_iCount].eType);
        _sTmp                     := Tc2_Standard.CONCAT(_sTmp, _sTab);
        _sTmp                     := Tc2_Standard.CONCAT(_sTmp, _aWriteList[_iCount].tTime);
        _sTmp                     := Tc2_Standard.CONCAT(_sTmp, _sTab);
        _sTmp                     := Tc2_Standard.CONCAT(_sTmp, Device_To_String(_aWriteList[_iCount].eDevice));
        _sTmp                     := Tc2_Standard.CONCAT(_sTmp, _sTab);
        _sTmp                     := Tc2_Standard.CONCAT(_sTmp, TO_STRING(_aWriteList[_iCount].eSubdevice));
        _sTmp                     := Tc2_Standard.CONCAT(_sTmp, _sTab);
        _sTmp                     := Tc2_Standard.CONCAT(_sTmp, TO_STRING(_aWriteList[_iCount].iErrorNumber));
        _sTmp                     := Tc2_Standard.CONCAT(_sTmp, _sTab);
        _sTmp                     := Tc2_Standard.CONCAT(_sTmp, _aWriteList[_iCount].sText);
        _sTmp                     := Tc2_Standard.CONCAT(_sTmp, _sNewLine);
        Builder(ADR(_sTmp), ADR(_sWriteData), StringLen(ADR(_sTmp)));
      END_IF
      _iCount                     := _iCount + 1;
  END_CASE
  CASE _eFlow
  OF
    E_MESSAGE_FLOW.MSG_FLOW_LINE_CHECK:
    IF NOT (_iCount > _iEnd)
    THEN
      _eFlow                      := E_MESSAGE_FLOW.MSG_FLOW_LINE_BUILD;
    ELSE
      _eState                     := E_PROGRESS.PROGRESS_WORKING;
      _eFlow                      := E_MESSAGE_FLOW.MSG_FLOW_WRITE_FILE_BUSY;
    END_IF
  END_CASE
END_CASE
//-----------------------------------------------------------------------------
//-----------------------------------------------------------------------------
CASE _eState
OF
  E_PROGRESS.PROGRESS_WORKING:
  CASE _eFlow
  OF
    E_MESSAGE_FLOW.MSG_FLOW_WRITE_FILE_BUSY:
      _nStringLength              := StringLen(ADR(_sWriteData));
      IF NOT (_nStringLength > 1)
      THEN
        _eState                   := E_PROGRESS.PROGRESS_DONE; 
       _eFlow                     := E_MESSAGE_FLOW.MSG_FLOW_WRITE_FILE_DONE;
      ELSE
        _eFlow                    := E_MESSAGE_FLOW.MSG_FLOW_WRITE_FILE_END;
        _eRes                     := WriteData(FALSE);
      END_IF
  END_CASE
  CASE _eFlow
  OF
    E_MESSAGE_FLOW.MSG_FLOW_WRITE_FILE_END:
      _eRes                       := WriteData(TRUE);

      IF (_eRes = E_PROGRESS.PROGRESS_ERROR)
      THEN
        _eState                   := E_PROGRESS.PROGRESS_ERROR;

      ELSIF (_eRes = E_PROGRESS.PROGRESS_DONE)
      THEN
        _eState                   := E_PROGRESS.PROGRESS_DONE;
        _eFlow                    := E_MESSAGE_FLOW.MSG_FLOW_WRITE_FILE_DONE;
        _eRes                     := WriteData(FALSE);
      END_IF
  END_CASE
END_CASE
//-----------------------------------------------------------------------------
//-----------------------------------------------------------------------------

BuildFileData                     := _eState;
END_METHOD

METHOD BuildFolder : e_progress
VAR_INPUT
  Execute           : BOOL;
END_VAR
VAR_INST
  _nErrorId   : UDINT;
  _eState     : E_PROGRESS;
  _eFlow      : E_MESSAGE_FLOW;
END_VAR
//-----------------------------------------------------------------------------
IF NOT Execute 
THEN 
	_eState                       := E_PROGRESS.PROGRESS_INIT; 
END_IF 
//-----------------------------------------------------------------------------
IF NOT Check() 
THEN 
	BuildFolder                   := E_PROGRESS.PROGRESS_ERROR; 
	RETURN; 
END_IF
//-----------------------------------------------------------------------------
//-----------------------------------------------------------------------------
CASE _eState
OF
  E_PROGRESS.PROGRESS_INIT:
    IF Execute
    THEN
      _nErrorId                 := 0;
      _bFileCreated             := FALSE;

      _sFolderDate              := FolderDate(_dtLocalTime);
      _eState                   := E_PROGRESS.PROGRESS_BUSY;
      _eFlow                    := E_MESSAGE_FLOW.MSG_FLOW_ROOT;
    END_IF
END_CASE
//-----------------------------------------------------------------------------
//-----------------------------------------------------------------------------
CASE _eState
OF
  E_PROGRESS.PROGRESS_BUSY:
  CASE _eFlow
  OF
    E_MESSAGE_FLOW.MSG_FLOW_ROOT:
      _eFlow                    := E_MESSAGE_FLOW.MSG_FLOW_ROOT_CREATE;
      _fbCreateDir.sPathName    := left(_pDirRoot^,len(_pDirRoot^)-1);
      _fbCreateDir(
              bExecute	        := FALSE);
    
    E_MESSAGE_FLOW.MSG_FLOW_ROOT_CREATE:
      (* create root folder *)
      _fbCreateDir(
              bExecute	        := TRUE);
      IF _fbCreateDir.bBusy
      THEN
        _eFlow                  := E_MESSAGE_FLOW.MSG_FLOW_ROOT_CREATE_BUSY;
      END_IF
    
    E_MESSAGE_FLOW.MSG_FLOW_ROOT_CREATE_BUSY:
      _fbCreateDir(
              bExecute	        := TRUE);
      IF NOT _fbCreateDir.bBusy
      THEN
        _eState                 := E_PROGRESS.PROGRESS_PREPARE;
        _eFlow                  := E_MESSAGE_FLOW.MSG_FLOW_FOLDER;
      END_IF
  END_CASE
END_CASE
//-----------------------------------------------------------------------------
//-----------------------------------------------------------------------------
CASE _eState
OF
  E_PROGRESS.PROGRESS_PREPARE:
  CASE _eFlow
  OF
    E_MESSAGE_FLOW.MSG_FLOW_FOLDER:
      _eFlow                    := E_MESSAGE_FLOW.MSG_FLOW_FOLDER_CREATE;
      _sFolderDate              := FolderDate(_dtLocalTime);
      _fbCreateDir.sPathName    := concat(_pDirRoot^, _sFolderDate);
      _fbCreateDir(
              bExecute	        := FALSE);
  
    E_MESSAGE_FLOW.MSG_FLOW_FOLDER_CREATE:
      (* create active folder *)
      _fbCreateDir(
              bExecute	        := TRUE);
      IF _fbCreateDir.bBusy
      THEN
        _eFlow                  := E_MESSAGE_FLOW.MSG_FLOW_FOLDER_CREATE_BUSY;
      END_IF
    
    E_MESSAGE_FLOW.MSG_FLOW_FOLDER_CREATE_BUSY:
      _fbCreateDir(
              bExecute	        := TRUE);
      IF NOT _fbCreateDir.bBusy
      THEN
        _eState                 := E_PROGRESS.PROGRESS_CHECK;
        _eFlow                  := E_MESSAGE_FLOW.MSG_FLOW_FILE_CREATE_DONE;
        _fbCreateDir(
                bExecute	      := FALSE);
      END_IF
  END_CASE
END_CASE
//-----------------------------------------------------------------------------
//-----------------------------------------------------------------------------
CASE _eState
OF
  E_PROGRESS.PROGRESS_CHECK:
  CASE _eFlow
  OF
    E_MESSAGE_FLOW.MSG_FLOW_FILE_CREATE_DONE:
      _eState                   := E_PROGRESS.PROGRESS_DONE;
      _bFileCreated             := TRUE;

      // build complete file path
      _sTmp                     := concat(concat(_pFileRoot^, _sFolderDate),'.txt');
      _sTmp                     := concat('\', _sTmp);
      _sFilename                := concat(_fbCreateDir.sPathName, _sTmp);
  END_CASE
END_CASE

BuildFolder                     := _eState;
END_METHOD

METHOD Check : BOOL
VAR_INPUT
END_VAR

IF NOT __ISVALIDREF(_stCtrl)
THEN
  _eCheck       := E_MESSAGE_CHECK.POINTER_CTRL_INVALID;
  RETURN;
END_IF

IF NOT __ISVALIDREF(_stState)
THEN
  _eCheck       := E_MESSAGE_CHECK.POINTER_STATE_INVALID;
  RETURN;
END_IF
//-----------------------------------------------------------------
//-----------------------------------------------------------------
IF NOT (_dtLocalTime <> 0)
THEN
  _eCheck       := E_MESSAGE_CHECK.POINTER_TIME_INVALID;
  RETURN;
END_IF

IF NOT (_pMsgList <> 0)
THEN
  _eCheck       := E_MESSAGE_CHECK.POINTER_LIST_INVALID;
  RETURN;
END_IF

IF NOT (_pFileRoot <> 0)
THEN
  _eCheck       := E_MESSAGE_CHECK.POINTER_ROOT_FILE_INVALID;
  RETURN;
END_IF

IF NOT (_pDirRoot <> 0)
THEN
  _eCheck       := E_MESSAGE_CHECK.POINTER_ROOT_DIR_INVALID;
  RETURN;
END_IF

IF NOT __ISVALIDREF(_nMsgIndex)
THEN
  _eCheck       := E_MESSAGE_CHECK.POINTER_MSG_IDX_INVALID;
  RETURN;
END_IF

IF NOT __ISVALIDREF(_nErrIndex)
THEN
  _eCheck       := E_MESSAGE_CHECK.POINTER_ERR_IDX_INVALID;
  RETURN;
END_IF


_eCheck         := E_MESSAGE_CHECK.CHECK_DONE;
Check           := TRUE;
END_METHOD

METHOD Cmd : e_message_state
VAR_INPUT
  Command     : e_message_ctrl;
END_VAR


CASE Command
OF
  E_MESSAGE_CTRL.MSG_CTRL_NULL:
    _eResult                    := E_PROGRESS.PROGRESS_INVALID;
    Cmd                         := E_MESSAGE_STATE.MSG_STATE_NULL;

  E_MESSAGE_CTRL.MSG_CTRL_INIT:
    _eResult                    := BuildFolder(FALSE);
    Cmd                         := E_MESSAGE_STATE.MSG_STATE_INIT;

  E_MESSAGE_CTRL.MSG_CTRL_IDLE:
    _eResult                    := BuildFileData(FALSE);
    Cmd                         := E_MESSAGE_STATE.MSG_STATE_IDLE;

  E_MESSAGE_CTRL.MSG_CTRL_WRITE:
    _eResult                    := BuildFileData(FALSE);
    Cmd                         := E_MESSAGE_STATE.MSG_STATE_WRITE;
    IF (_nMsgIndex = 0)
    THEN
       // go back to sleep
      _eResult                := E_PROGRESS.PROGRESS_DONE;
    END_IF
ELSE
    //_eResult                    := E_PROGRESS.PROGRESS_ERROR;
    Cmd                         := E_MESSAGE_STATE.MSG_STATE_NULL;
END_CASE
END_METHOD

PROPERTY Ctrl : REFERENCE to ST_MESSAGE_CTRL
SET
_stCtrl ref= Ctrl;
END_SET
END_PROPERTY

PROPERTY FileCreated : bool
GET
FileCreated := _bFileCreated;
END_GET
END_PROPERTY

PROPERTY State : REFERENCE TO ST_MESSAGE_STATE
SET
_stState ref= State;
END_SET
END_PROPERTY

END_FUNCTION_BLOCK

// ---- APPLICATION/MAIN_APP.TcPOU
//---------------------------------------------------------------------------------------------------------------
//
//  HAUD 2026.03.21
//
//  - MAIN_APPLICATION helper
//    - example PRG for setting up your application startup
//
//---------------------------------------------------------------------------------------------------------------
// This SOFTWARE is provided as an Example by THE PROVIDER "as is" and "with all faults." THE PROVIDER makes no 
// representations or warranties of any kind concerning the safety, suitability, lack of viruses, inaccuracies, 
// typographical errors, or other harmful components of this SOFTWARE. There are inherent dangers in the use of 
// any software, and you are solely responsible for determining whether this SOFTWARE is compatible with your 
// equipment and other software installed on your equipment. You are also solely responsible for the protection 
// of your equipment and backup of your data, and THE PROVIDER will not be liable for any damages you may suffer 
// in connection with using, modifying, or distributing this SOFTWARE.
//---------------------------------------------------------------------------------------------------------------
PROGRAM MAIN_APP
VAR
  eInit      AT %Q*     : E_PROGRESS;   // startup state machine after MAIN is initialized
  bXmlStartup           : BOOL;         // optional example switch for using xml configuration
END_VAR

//-----------------------------------------------------------------------------
// wait for initialization to be complete before work may start
//-----------------------------------------------------------------------------
IF NOT (MAIN_XTS.eInit = E_PROGRESS.PROGRESS_DONE)
THEN
  eInit                                       := E_PROGRESS.PROGRESS_INIT;
  RETURN;
END_IF
//-----------------------------------------------------------------------------
//-----------------------------------------------------------------------------
// start your application init from here (example)
//-----------------------------------------------------------------------------
CASE eInit
OF
  //---------------------------------------------------------------------------
  E_PROGRESS.PROGRESS_NOT_EXIST:
    RETURN;       // you just bypassed the mapping
                  // check if you require anything from the initialisation
  //---------------------------------------------------------------------------
  E_PROGRESS.PROGRESS_INIT:
    GVL_APPLICATION.ConfigCtrl.Cmd            := E_DATA_CTRL.NULL;
    eInit                                     := E_PROGRESS.PROGRESS_BUSY;

  //---------------------------------------------------------------------------
  E_PROGRESS.PROGRESS_BUSY:
    IF NOT bXmlStartup
    THEN
      StationParameterExample();
      eInit                                   := E_PROGRESS.PROGRESS_WORKING;
    ELSE
      GVL_APPLICATION.ConfigCtrl.Cmd          := E_DATA_CTRL.INIT;
      eInit                                   := E_PROGRESS.PROGRESS_PREPARE;
    END_IF

  //---------------------------------------------------------------------------
  E_PROGRESS.PROGRESS_PREPARE:
    IF (GVL_APPLICATION.ConfigState.State = E_DATA_STATE.INIT + E_PROGRESS.PROGRESS_DONE)
    THEN
      GVL_APPLICATION.ConfigCtrl.Cmd          := E_DATA_CTRL.READ;
      eInit                                   := E_PROGRESS.PROGRESS_STARTUP;
    END_IF

  E_PROGRESS.PROGRESS_STARTUP:
    IF (GVL_APPLICATION.ConfigState.State = E_DATA_STATE.READ + E_PROGRESS.PROGRESS_DONE)
    THEN
      GVL_APPLICATION.ConfigCtrl.Cmd          := E_DATA_CTRL.NULL;
      eInit                                   := E_PROGRESS.PROGRESS_CHECK;
    END_IF

  E_PROGRESS.PROGRESS_CHECK:
    eInit                                     := E_PROGRESS.PROGRESS_OCCUPIED;

  E_PROGRESS.PROGRESS_OCCUPIED:
    eInit                                     := E_PROGRESS.PROGRESS_WORKING;

  E_PROGRESS.PROGRESS_WORKING:
    eInit                                     := E_PROGRESS.PROGRESS_DONE;
END_CASE
//-----------------------------------------------------------------------------
//-----------------------------------------------------------------------------
//-----------------------------------------------------------------------------
// connect data and control to xml configuration
GVL_APPLICATION.StationConfig.Identity        :=   GVL_XTS.Xpu.XpuOtcid;
GVL_APPLICATION.StationConfig.Ctrl            REF= GVL_APPLICATION.ConfigCtrl;
GVL_APPLICATION.StationConfig.State           REF= GVL_APPLICATION.ConfigState;

GVL_APPLICATION.StationConfig.MessageDevice   := e_Device.Device_Configuration;
GVL_APPLICATION.StationConfig.MessageLevel    := GVL_MSG_XTS.MessageLevel;
GVL_APPLICATION.StationConfig.FolderPath      := GVL_MSG_XTS.CON_DIR;
GVL_APPLICATION.StationConfig.StationParameter:= ADR(GVL_XTS.StationParameter);

GVL_APPLICATION.StationConfig();        // call xml configuration
//-----------------------------------------------------------------------------
//-----------------------------------------------------------------------------

END_PROGRAM

// ---- APPLICATION/StationParameterExample.TcPOU
FUNCTION StationParameterExample  : BOOL
VAR
  nStationParameter                 : UINT; // THIS IS ONLY FOR EXAMPLE USE, CHECK MAX_STATION MANUALLY
END_VAR

//-----------------------------------------------------------------------------------------------------------------------------------------
//-----------------------------------------------------------------------------------------------------------------------------------------
//
//  HAUD 2026.05.26
//
//  - hard coded station parameters as example
//  - TODO: xml DataServer implementation for station parameter read/write
//
//  - reminder: (this you HAVE to check manually when setting up the transport)
//-----------------------------------------------------------------------------
//    - DO NOT place the modulo turn within the range of a station
//
//    - in case the extern process requires multiple xts stations, 
//      - the range must be closed and in strict order
//-----------------------------------------------------------------------------------------------------------------------------------------
//-----------------------------------------------------------------------------------------------------------------------------------------
GVL_XTS.StationStartIndex                                         := 2;
GVL_XTS.StationStart.rPosWait                                     :=    125.0; // for every TRANSPORT_START this physical position may differ from the rPosWait of StationStartIndex station

GVL_XTS.StationStart.rGap                                         :=    175.0;
GVL_XTS.StationStart.rVelo                                        :=   1250.0;
GVL_XTS.StationStart.rAccDec                                      :=  17500.0;
GVL_XTS.StationStart.rJerk                                        := 600000.0;
//-----------------------------------------------------------------------------------------------------------------------------------------
// THIS IS ONLY FOR EXAMPLE USE, 
//  CHECK GVL_XTS.MAX_STATION MANUALLY
//-----------------------------------------------------------------------------------------------------------------------------------------
nStationParameter := 1;
GVL_XTS.StationParameter[nStationParameter].eType                 := E_STATION_TYPE.STATION_PROCESS;
GVL_XTS.StationParameter[nStationParameter].sText                 := concat('DIST_0', TO_STRING(nStationParameter));
GVL_XTS.StationParameter[nStationParameter].rPosWait              :=  21000.0; // absolute modulo position

GVL_XTS.StationParameter[nStationParameter].nConfiguredStopCount  :=      1;   // how many stops the mover has to make in this station
GVL_XTS.StationParameter[nStationParameter].rPosStop[1]           :=      0.0; // relative to rPosWait

GVL_XTS.StationParameter[nStationParameter].rReleaseDistance      :=     -5.0; // relative to Mover.ActPos

GVL_XTS.StationParameter[nStationParameter].rGap                  :=    150.0;
GVL_XTS.StationParameter[nStationParameter].rVelo                 :=   1250.0;
GVL_XTS.StationParameter[nStationParameter].rAccDec               :=  17500.0;
GVL_XTS.StationParameter[nStationParameter].rJerk                 := 600000.0;
//-----------------------------------------------------------------------------------------------------------------------------------------
// THIS IS ONLY FOR EXAMPLE USE, 
//  CHECK GVL_XTS.MAX_STATION MANUALLY
//-----------------------------------------------------------------------------------------------------------------------------------------
nStationParameter := 2;
GVL_XTS.StationParameter[nStationParameter].eType                 := E_STATION_TYPE.STATION_PROCESS;
GVL_XTS.StationParameter[nStationParameter].sText                 := concat('DIST_0', TO_STRING(nStationParameter));
GVL_XTS.StationParameter[nStationParameter].rPosWait              :=    500.0; // absolute modulo position

GVL_XTS.StationParameter[nStationParameter].nConfiguredStopCount  :=      1;   // how many stops the mover has to make in this station
GVL_XTS.StationParameter[nStationParameter].rPosStop[1]           :=      0.0; // relative to rPosWait

GVL_XTS.StationParameter[nStationParameter].rReleaseDistance      :=     -5.0; // relative to Mover.ActPos

GVL_XTS.StationParameter[nStationParameter].rGap                  :=    105.0;
GVL_XTS.StationParameter[nStationParameter].rVelo                 :=   2500.0;
GVL_XTS.StationParameter[nStationParameter].rAccDec               :=  17500.0;
GVL_XTS.StationParameter[nStationParameter].rJerk                 := 600000.0;
//-----------------------------------------------------------------------------------------------------------------------------------------
// THIS IS ONLY FOR EXAMPLE USE, 
//  CHECK GVL_XTS.MAX_STATION MANUALLY
//-----------------------------------------------------------------------------------------------------------------------------------------
nStationParameter := 3;
GVL_XTS.StationParameter[nStationParameter].eType                 := E_STATION_TYPE.STATION_PROCESS;
GVL_XTS.StationParameter[nStationParameter].sText                 := concat('STN_0', TO_STRING(nStationParameter*10));
GVL_XTS.StationParameter[nStationParameter].rPosWait              :=   2000.0; // absolute modulo position

GVL_XTS.StationParameter[nStationParameter].nConfiguredStopCount  :=      2;   // how many stops the mover has to make in this station
GVL_XTS.StationParameter[nStationParameter].rPosStop[1]           :=    700.0; // relative to rPosWait
GVL_XTS.StationParameter[nStationParameter].rPosStop[2]           :=    850.0; // relative to rPosWait

GVL_XTS.StationParameter[nStationParameter].rReleaseDistance      :=     25.0; // relative to Mover.ActPos

GVL_XTS.StationParameter[nStationParameter].rGap                  :=    105.0;
GVL_XTS.StationParameter[nStationParameter].rVelo                 :=   2500.0;
GVL_XTS.StationParameter[nStationParameter].rAccDec               :=  17500.0;
GVL_XTS.StationParameter[nStationParameter].rJerk                 := 600000.0;
//-----------------------------------------------------------------------------------------------------------------------------------------
// THIS IS ONLY FOR EXAMPLE USE, 
//  CHECK GVL_XTS.MAX_STATION MANUALLY
//-----------------------------------------------------------------------------------------------------------------------------------------
nStationParameter := 4;
GVL_XTS.StationParameter[nStationParameter].eType                 := E_STATION_TYPE.STATION_PROCESS;
GVL_XTS.StationParameter[nStationParameter].sText                 := 'STN_060';
GVL_XTS.StationParameter[nStationParameter].rPosWait              :=    5000.0; // absolute modulo position

GVL_XTS.StationParameter[nStationParameter].nConfiguredStopCount  :=      1;   // how many stops the mover has to make in this station
GVL_XTS.StationParameter[nStationParameter].rPosStop[1]           :=    500.0; // relative to rPosWait

GVL_XTS.StationParameter[nStationParameter].rReleaseDistance      :=    300.0; // relative to Mover.ActPos

GVL_XTS.StationParameter[nStationParameter].rGap                  :=    105.0;
GVL_XTS.StationParameter[nStationParameter].rVelo                 :=   2500.0;
GVL_XTS.StationParameter[nStationParameter].rAccDec               :=  17500.0;
GVL_XTS.StationParameter[nStationParameter].rJerk                 := 600000.0;

nStationParameter := 5;
GVL_XTS.StationParameter[nStationParameter].eType                 := E_STATION_TYPE.STATION_PROCESS;
GVL_XTS.StationParameter[nStationParameter].sText                 := 'STN_060';
GVL_XTS.StationParameter[nStationParameter].rPosWait              :=    5000.0; // absolute modulo position

GVL_XTS.StationParameter[nStationParameter].nConfiguredStopCount  :=      1;   // how many stops the mover has to make in this station
GVL_XTS.StationParameter[nStationParameter].rPosStop[1]           :=    850.0; // relative to rPosWait

GVL_XTS.StationParameter[nStationParameter].rReleaseDistance      :=     25.0; // relative to Mover.ActPos

GVL_XTS.StationParameter[nStationParameter].rGap                  :=    105.0;
GVL_XTS.StationParameter[nStationParameter].rVelo                 :=   2500.0;
GVL_XTS.StationParameter[nStationParameter].rAccDec               :=  17500.0;
GVL_XTS.StationParameter[nStationParameter].rJerk                 := 600000.0;
//-----------------------------------------------------------------------------------------------------------------------------------------
// THIS IS ONLY FOR EXAMPLE USE, 
//  CHECK GVL_XTS.MAX_STATION MANUALLY
//-----------------------------------------------------------------------------------------------------------------------------------------
nStationParameter := 6;
GVL_XTS.StationParameter[nStationParameter].eType                 := E_STATION_TYPE.STATION_PROCESS;
GVL_XTS.StationParameter[nStationParameter].sText                 := 'STN_070';
GVL_XTS.StationParameter[nStationParameter].rPosWait              :=   6000.0; // absolute modulo position

GVL_XTS.StationParameter[nStationParameter].nConfiguredStopCount  :=      1;   // how many stops the mover has to make in this station
GVL_XTS.StationParameter[nStationParameter].rPosStop[1]           :=    500.0; // relative to rPosWait

GVL_XTS.StationParameter[nStationParameter].rReleaseDistance      :=    300.0; // relative to Mover.ActPos

GVL_XTS.StationParameter[nStationParameter].rGap                  :=    105.0;
GVL_XTS.StationParameter[nStationParameter].rVelo                 :=   2500.0;
GVL_XTS.StationParameter[nStationParameter].rAccDec               :=  17500.0;
GVL_XTS.StationParameter[nStationParameter].rJerk                 := 600000.0;

nStationParameter := 7;
GVL_XTS.StationParameter[nStationParameter].eType                 := E_STATION_TYPE.STATION_PROCESS;
GVL_XTS.StationParameter[nStationParameter].sText                 := 'STN_070';
GVL_XTS.StationParameter[nStationParameter].rPosWait              :=   6000.0; // absolute modulo position

GVL_XTS.StationParameter[nStationParameter].nConfiguredStopCount  :=      1;   // how many stops the mover has to make in this station
GVL_XTS.StationParameter[nStationParameter].rPosStop[1]           :=    850.0; // relative to rPosWait

GVL_XTS.StationParameter[nStationParameter].rReleaseDistance      :=     25.0; // relative to Mover.ActPos

GVL_XTS.StationParameter[nStationParameter].rGap                  :=    105.0;
GVL_XTS.StationParameter[nStationParameter].rVelo                 :=   2500.0;
GVL_XTS.StationParameter[nStationParameter].rAccDec               :=  17500.0;
GVL_XTS.StationParameter[nStationParameter].rJerk                 := 600000.0;
//-----------------------------------------------------------------------------------------------------------------------------------------
// THIS IS ONLY FOR EXAMPLE USE, 
//  CHECK GVL_XTS.MAX_STATION MANUALLY
//-----------------------------------------------------------------------------------------------------------------------------------------
nStationParameter := 8;
GVL_XTS.StationParameter[nStationParameter].eType                 := E_STATION_TYPE.STATION_PROCESS;
GVL_XTS.StationParameter[nStationParameter].sText                 := 'STN_100';
GVL_XTS.StationParameter[nStationParameter].rPosWait              :=   9000.0; // absolute modulo position

GVL_XTS.StationParameter[nStationParameter].nConfiguredStopCount  :=      2;   // how many stops the mover has to make in this station
GVL_XTS.StationParameter[nStationParameter].rPosStop[1]           :=    500.0; // relative to rPosWait
GVL_XTS.StationParameter[nStationParameter].rPosStop[1]           :=    550.0; // relative to rPosWait

GVL_XTS.StationParameter[nStationParameter].rReleaseDistance      :=     25.0; // relative to Mover.ActPos

GVL_XTS.StationParameter[nStationParameter].rGap                  :=    105.0;
GVL_XTS.StationParameter[nStationParameter].rVelo                 :=   2500.0;
GVL_XTS.StationParameter[nStationParameter].rAccDec               :=  17500.0;
GVL_XTS.StationParameter[nStationParameter].rJerk                 := 600000.0;
//-----------------------------------------------------------------------------------------------------------------------------------------
// THIS IS ONLY FOR EXAMPLE USE, 
//  CHECK GVL_XTS.MAX_STATION MANUALLY
//-----------------------------------------------------------------------------------------------------------------------------------------
nStationParameter := 9;
GVL_XTS.StationParameter[nStationParameter].eType                 := E_STATION_TYPE.STATION_PROCESS;
GVL_XTS.StationParameter[nStationParameter].sText                 := 'DIST_100';
GVL_XTS.StationParameter[nStationParameter].rPosWait              :=   10000.0; // absolute modulo position

GVL_XTS.StationParameter[nStationParameter].nConfiguredStopCount  :=      1;   // how many stops the mover has to make in this station
GVL_XTS.StationParameter[nStationParameter].rPosStop[1]           :=      0.0; // relative to rPosWait
GVL_XTS.StationParameter[nStationParameter].rPosStop[1]           :=      0.0; // relative to rPosWait

GVL_XTS.StationParameter[nStationParameter].rReleaseDistance      :=     -5.0; // relative to Mover.ActPos

GVL_XTS.StationParameter[nStationParameter].rGap                  :=    150.0;
GVL_XTS.StationParameter[nStationParameter].rVelo                 :=   1250.0;
GVL_XTS.StationParameter[nStationParameter].rAccDec               :=  17500.0;
GVL_XTS.StationParameter[nStationParameter].rJerk                 := 600000.0;
//-----------------------------------------------------------------------------------------------------------------------------------------
// THIS IS ONLY FOR EXAMPLE USE, 
//  CHECK GVL_XTS.MAX_STATION MANUALLY
//-----------------------------------------------------------------------------------------------------------------------------------------
nStationParameter := 10;
GVL_XTS.StationParameter[nStationParameter].eType                 := E_STATION_TYPE.STATION_PROCESS;
GVL_XTS.StationParameter[nStationParameter].sText                 := 'STN_110';
GVL_XTS.StationParameter[nStationParameter].rPosWait              :=   11000.0; // absolute modulo position

GVL_XTS.StationParameter[nStationParameter].nConfiguredStopCount  :=      1;   // how many stops the mover has to make in this station
GVL_XTS.StationParameter[nStationParameter].rPosStop[1]           :=    700.0; // relative to rPosWait

GVL_XTS.StationParameter[nStationParameter].rReleaseDistance      :=    150.0; // relative to Mover.ActPos

GVL_XTS.StationParameter[nStationParameter].rGap                  :=    105.0;
GVL_XTS.StationParameter[nStationParameter].rVelo                 :=   2500.0;
GVL_XTS.StationParameter[nStationParameter].rAccDec               :=  17500.0;
GVL_XTS.StationParameter[nStationParameter].rJerk                 := 600000.0;

